// TIA Portal V17 export
// export: Created 2024-09-02T12:50:15.4689552Z, ExportSetting WithDefaults, DisplayName Totally Integrated Automation Portal, DisplayVersion V17, DisplayName TIA Portal Openness, DisplayVersion V17, DisplayName TIA Portal Version Control Interface, DisplayVersion V17, DisplayName STEP 7 Professional, DisplayVersion V17, DisplayName STEP 7 Safety, DisplayVersion V17, DisplayName WinCC Professional, DisplayVersion V17
FUNCTION "AnwFC_ZP_HMI_Management_OP70" : Void   // FC59, LAD
TITLE = HMI supply / HMI Versorgung
{ S7_Optimized_Access := 'TRUE' }
AUTHOR : OlegFuehrus
FAMILY : BA
NAME : BA
VERSION : 0.1
// stored: AutoNumber true, IsIECCheckEnabled false, SetENOAutomatically false, UDAEnableTagReadback false
   VAR_TEMP
      t_StationReady : Bool;
      tTyp : Int;
   END_VAR
   VAR_TEMP   // added for the SCL form of the ladder/FBD networks
      _w1 : Bool;
      _w2 : Bool;
   END_VAR
BEGIN

REGION Network 1: Image selection: Basic screen / Bildanwahl: Grundbild
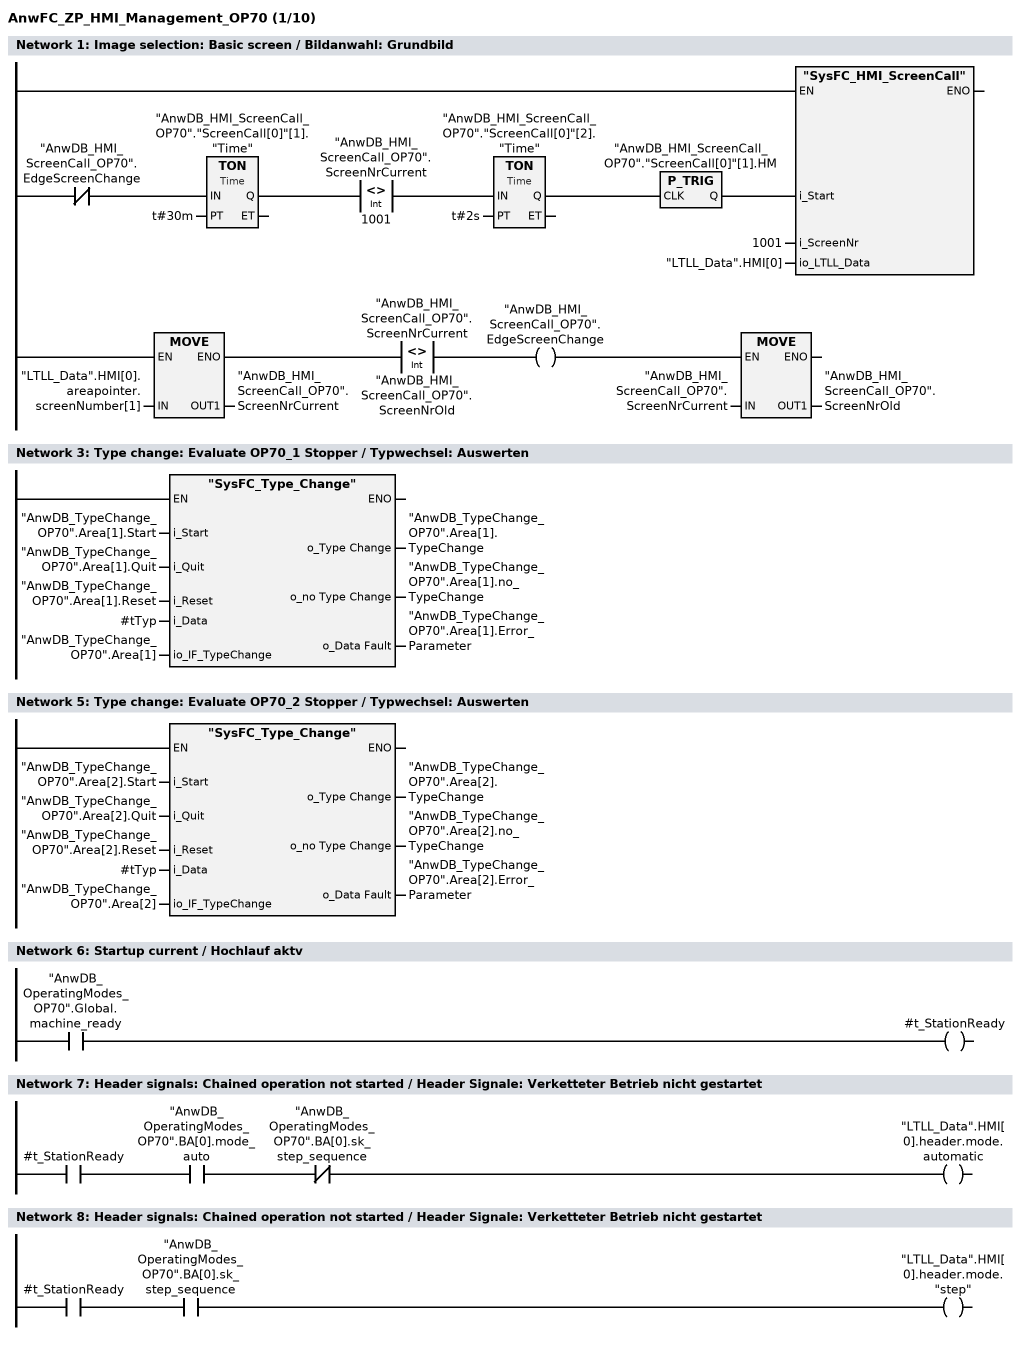
   RUNG wire#powerrail
      "SysFC_HMI_ScreenCall"(i_Start := wire#w1, i_ScreenNr := 1001, io_LTLL_Data := "LTLL_Data".HMI[0])
   END_RUNG
   RUNG wire#powerrail
      I_Contact( "AnwDB_HMI_ScreenCall_OP70".EdgeScreenChange )
      { S7_Templates := "time_type := Time" } "AnwDB_HMI_ScreenCall_OP70"."ScreenCall[0]"[1]."Time".TON(pt := t#30m, et =>)
      { S7_Templates := "SrcType := Int" } NE_Contact(in1 := "AnwDB_HMI_ScreenCall_OP70".ScreenNrCurrent, in2 := 1001)
      { S7_Templates := "time_type := Time" } "AnwDB_HMI_ScreenCall_OP70"."ScreenCall[0]"[2]."Time".TON(pt := t#2s, et =>)
      P_Trig( "AnwDB_HMI_ScreenCall_OP70"."ScreenCall[0]"[1].HM )
   END_RUNG wire#w1
   RUNG wire#powerrail
      Move(in := "LTLL_Data".HMI[0].areapointer.screenNumber[1], out1 => "AnwDB_HMI_ScreenCall_OP70".ScreenNrCurrent)
      { S7_Templates := "SrcType := Int" } NE_Contact(in1 := "AnwDB_HMI_ScreenCall_OP70".ScreenNrCurrent, in2 := "AnwDB_HMI_ScreenCall_OP70".ScreenNrOld)
      Coil( "AnwDB_HMI_ScreenCall_OP70".EdgeScreenChange )
      Move(in := "AnwDB_HMI_ScreenCall_OP70".ScreenNrCurrent, out1 => "AnwDB_HMI_ScreenCall_OP70".ScreenNrOld)
   END_RUNG
   // the same network as SCL:
   "AnwDB_HMI_ScreenCall_OP70"."ScreenCall[0]"[1]."Time".TON(IN := NOT "AnwDB_HMI_ScreenCall_OP70".EdgeScreenChange,
                           PT := t#30m);
   "AnwDB_HMI_ScreenCall_OP70"."ScreenCall[0]"[2]."Time".TON(IN := "AnwDB_HMI_ScreenCall_OP70"."ScreenCall[0]"[1]."Time".Q AND ("AnwDB_HMI_ScreenCall_OP70".ScreenNrCurrent <> 1001),
                           PT := t#2s);
   #_w1 := "AnwDB_HMI_ScreenCall_OP70"."ScreenCall[0]"[2]."Time".Q;
   #_w2 := #_w1 AND NOT "AnwDB_HMI_ScreenCall_OP70"."ScreenCall[0]"[1].HM;   // rising edge
   "AnwDB_HMI_ScreenCall_OP70"."ScreenCall[0]"[1].HM := #_w1;
   "SysFC_HMI_ScreenCall"(i_Start := #_w2, i_ScreenNr := 1001, io_LTLL_Data := "LTLL_Data".HMI[0]);
   "AnwDB_HMI_ScreenCall_OP70".ScreenNrCurrent := "LTLL_Data".HMI[0].areapointer.screenNumber[1];
   "AnwDB_HMI_ScreenCall_OP70".EdgeScreenChange := "AnwDB_HMI_ScreenCall_OP70".ScreenNrCurrent <> "AnwDB_HMI_ScreenCall_OP70".ScreenNrOld;
   IF "AnwDB_HMI_ScreenCall_OP70".EdgeScreenChange THEN
       "AnwDB_HMI_ScreenCall_OP70".ScreenNrOld := "AnwDB_HMI_ScreenCall_OP70".ScreenNrCurrent;
   END_IF;
END_REGION

REGION Network 2 (SCL): Type change: Copy type no. OP70_1 Stopper / Typwechsel: Typ-Nr. kopieren
   #tTyp := "MdsDB1_FG01_Data_SLG1_OP70".read.General."Variant Number";
END_REGION

REGION Network 3: Type change: Evaluate OP70_1 Stopper / Typwechsel: Auswerten
   RUNG wire#powerrail
      "SysFC_Type_Change"(i_Start := "AnwDB_TypeChange_OP70".Area[1].Start, i_Quit := "AnwDB_TypeChange_OP70".Area[1].Quit, i_Reset := "AnwDB_TypeChange_OP70".Area[1].Reset, i_Data := #tTyp, io_IF_TypeChange := "AnwDB_TypeChange_OP70".Area[1], "o_Type Change" => "AnwDB_TypeChange_OP70".Area[1].TypeChange, "o_no Type Change" => "AnwDB_TypeChange_OP70".Area[1].no_TypeChange, "o_Data Fault" => "AnwDB_TypeChange_OP70".Area[1].Error_Parameter)
   END_RUNG
   // the same network as SCL:
   "SysFC_Type_Change"(i_Start := "AnwDB_TypeChange_OP70".Area[1].Start,
                       i_Quit := "AnwDB_TypeChange_OP70".Area[1].Quit,
                       i_Reset := "AnwDB_TypeChange_OP70".Area[1].Reset,
                       i_Data := #tTyp,
                       io_IF_TypeChange := "AnwDB_TypeChange_OP70".Area[1],
                       "o_Type Change" => "AnwDB_TypeChange_OP70".Area[1].TypeChange,
                       "o_no Type Change" => "AnwDB_TypeChange_OP70".Area[1].no_TypeChange,
                       "o_Data Fault" => "AnwDB_TypeChange_OP70".Area[1].Error_Parameter);
END_REGION

REGION Network 4 (SCL): Type change: Copy type no. OP70_2 Stopper / Typwechsel: Typ-Nr. kopieren
   #tTyp := "MdsDB1_FG02_Data_SLG3_OP70".read.General."Variant Number";
END_REGION

REGION Network 5: Type change: Evaluate OP70_2 Stopper / Typwechsel: Auswerten
   RUNG wire#powerrail
      "SysFC_Type_Change"(i_Start := "AnwDB_TypeChange_OP70".Area[2].Start, i_Quit := "AnwDB_TypeChange_OP70".Area[2].Quit, i_Reset := "AnwDB_TypeChange_OP70".Area[2].Reset, i_Data := #tTyp, io_IF_TypeChange := "AnwDB_TypeChange_OP70".Area[2], "o_Type Change" => "AnwDB_TypeChange_OP70".Area[2].TypeChange, "o_no Type Change" => "AnwDB_TypeChange_OP70".Area[2].no_TypeChange, "o_Data Fault" => "AnwDB_TypeChange_OP70".Area[2].Error_Parameter)
   END_RUNG
   // the same network as SCL:
   "SysFC_Type_Change"(i_Start := "AnwDB_TypeChange_OP70".Area[2].Start,
                       i_Quit := "AnwDB_TypeChange_OP70".Area[2].Quit,
                       i_Reset := "AnwDB_TypeChange_OP70".Area[2].Reset,
                       i_Data := #tTyp,
                       io_IF_TypeChange := "AnwDB_TypeChange_OP70".Area[2],
                       "o_Type Change" => "AnwDB_TypeChange_OP70".Area[2].TypeChange,
                       "o_no Type Change" => "AnwDB_TypeChange_OP70".Area[2].no_TypeChange,
                       "o_Data Fault" => "AnwDB_TypeChange_OP70".Area[2].Error_Parameter);
END_REGION

REGION Network 6: Startup current / Hochlauf aktv
   RUNG wire#powerrail
      Contact( "AnwDB_OperatingModes_OP70".Global.machine_ready )
      Coil( #t_StationReady )
   END_RUNG
   // the same network as SCL:
   #t_StationReady := "AnwDB_OperatingModes_OP70".Global.machine_ready;
END_REGION

REGION Network 7: Header signals: Chained operation not started / Header Signale: Verketteter Betrieb nicht gestartet
   RUNG wire#powerrail
      Contact( #t_StationReady )
      Contact( "AnwDB_OperatingModes_OP70".BA[0].mode_auto )
      I_Contact( "AnwDB_OperatingModes_OP70".BA[0].sk_step_sequence )
      Coil( "LTLL_Data".HMI[0].header.mode.automatic )
   END_RUNG
   // the same network as SCL:
   "LTLL_Data".HMI[0].header.mode.automatic := #t_StationReady AND "AnwDB_OperatingModes_OP70".BA[0].mode_auto AND NOT "AnwDB_OperatingModes_OP70".BA[0].sk_step_sequence;
END_REGION

REGION Network 8: Header signals: Chained operation not started / Header Signale: Verketteter Betrieb nicht gestartet
   RUNG wire#powerrail
      Contact( #t_StationReady )
      Contact( "AnwDB_OperatingModes_OP70".BA[0].sk_step_sequence )
      Coil( "LTLL_Data".HMI[0].header.mode."step" )
   END_RUNG
   // the same network as SCL:
   "LTLL_Data".HMI[0].header.mode."step" := #t_StationReady AND "AnwDB_OperatingModes_OP70".BA[0].sk_step_sequence;
END_REGION

REGION Network 9: Header signals: Setup mode / Header Signale: Einrichtbetrieb
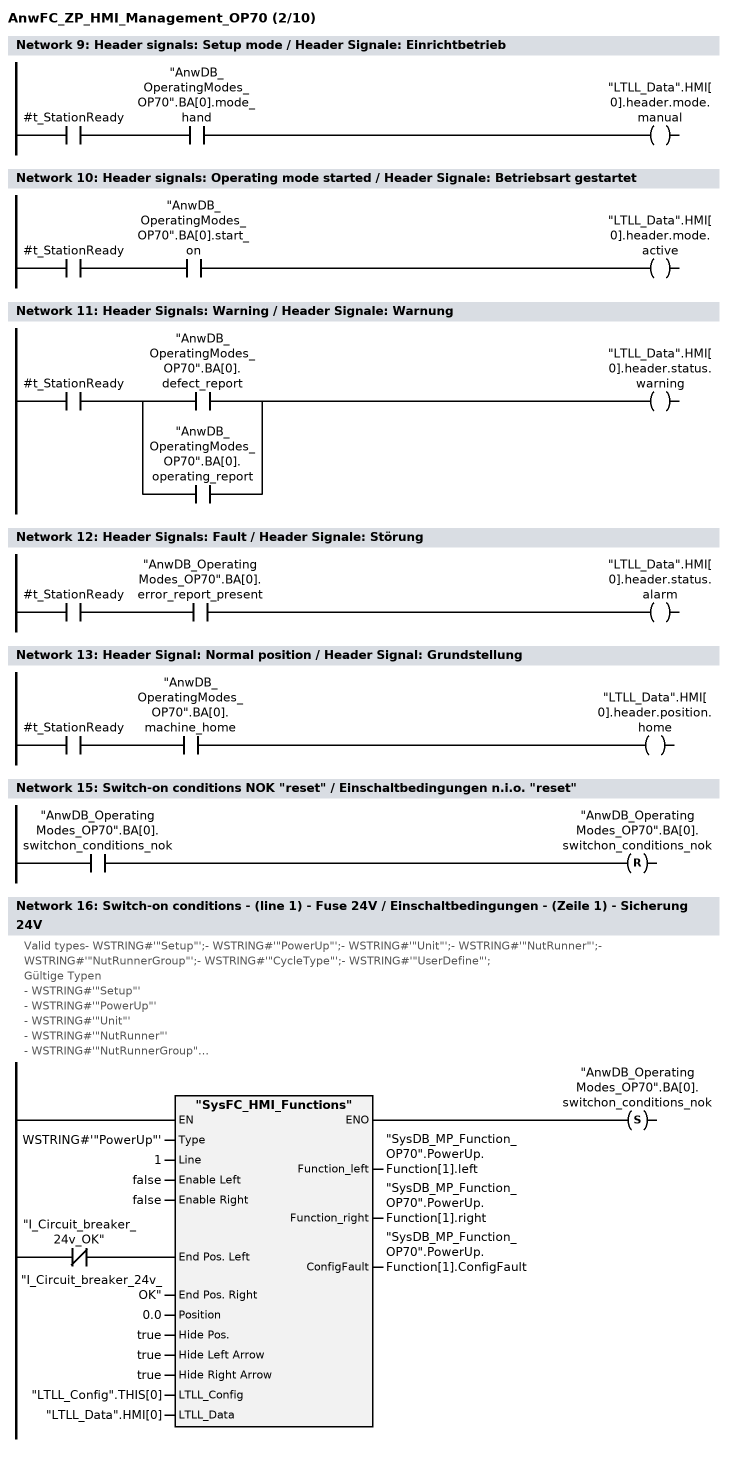
   RUNG wire#powerrail
      Contact( #t_StationReady )
      Contact( "AnwDB_OperatingModes_OP70".BA[0].mode_hand )
      Coil( "LTLL_Data".HMI[0].header.mode.manual )
   END_RUNG
   // the same network as SCL:
   "LTLL_Data".HMI[0].header.mode.manual := #t_StationReady AND "AnwDB_OperatingModes_OP70".BA[0].mode_hand;
END_REGION

REGION Network 10: Header signals: Operating mode started / Header Signale: Betriebsart gestartet
   RUNG wire#powerrail
      Contact( #t_StationReady )
      Contact( "AnwDB_OperatingModes_OP70".BA[0].start_on )
      Coil( "LTLL_Data".HMI[0].header.mode.active )
   END_RUNG
   // the same network as SCL:
   "LTLL_Data".HMI[0].header.mode.active := #t_StationReady AND "AnwDB_OperatingModes_OP70".BA[0].start_on;
END_REGION

REGION Network 11: Header Signals: Warning / Header Signale: Warnung
   RUNG wire#powerrail
      Contact( #t_StationReady )
      wire#w1
      Contact( "AnwDB_OperatingModes_OP70".BA[0].defect_report )
      wire#w2
      Coil( "LTLL_Data".HMI[0].header.status.warning )
   END_RUNG
   RUNG wire#w1
      Contact( "AnwDB_OperatingModes_OP70".BA[0].operating_report )
   END_RUNG wire#w2
   // the same network as SCL:
   "LTLL_Data".HMI[0].header.status.warning := #t_StationReady AND ("AnwDB_OperatingModes_OP70".BA[0].defect_report OR "AnwDB_OperatingModes_OP70".BA[0].operating_report);
END_REGION

REGION Network 12: Header Signals: Fault / Header Signale: Störung
   RUNG wire#powerrail
      Contact( #t_StationReady )
      Contact( "AnwDB_OperatingModes_OP70".BA[0].error_report_present )
      Coil( "LTLL_Data".HMI[0].header.status.alarm )
   END_RUNG
   // the same network as SCL:
   "LTLL_Data".HMI[0].header.status.alarm := #t_StationReady AND "AnwDB_OperatingModes_OP70".BA[0].error_report_present;
END_REGION

REGION Network 13: Header Signal: Normal position / Header Signal: Grundstellung
   RUNG wire#powerrail
      Contact( #t_StationReady )
      Contact( "AnwDB_OperatingModes_OP70".BA[0].machine_home )
      Coil( "LTLL_Data".HMI[0].header.position.home )
   END_RUNG
   // the same network as SCL:
   "LTLL_Data".HMI[0].header.position.home := #t_StationReady AND "AnwDB_OperatingModes_OP70".BA[0].machine_home;
END_REGION

REGION Network 14: ############# SO_02_002_PowerUpCondition ############## / ######################## SS_02_002_PowerUpCondition #########################
END_REGION

REGION Network 15: Switch-on conditions NOK "reset" / Einschaltbedingungen n.i.o. "reset"
   RUNG wire#powerrail
      Contact( "AnwDB_OperatingModes_OP70".BA[0].switchon_conditions_nok )
      R_Coil( "AnwDB_OperatingModes_OP70".BA[0].switchon_conditions_nok )
   END_RUNG
   // the same network as SCL:
   IF "AnwDB_OperatingModes_OP70".BA[0].switchon_conditions_nok THEN
       "AnwDB_OperatingModes_OP70".BA[0].switchon_conditions_nok := FALSE;
   END_IF;
END_REGION

REGION Network 16: Switch-on conditions - (line 1) - Fuse 24V / Einschaltbedingungen - (Zeile 1) - Sicherung 24V
   // Valid types- WSTRING#'"Setup"';- WSTRING#'"PowerUp"';- WSTRING#'"Unit"';- WSTRING#'"NutRunner"';- WSTRING#'"NutRunnerGroup"';- WSTRING#'"CycleType"';- WSTRING#'"UserDefine"';
   // Gültige Typen
   // - WSTRING#'"Setup"'
   // - WSTRING#'"PowerUp"'
   // - WSTRING#'"Unit"'
   // - WSTRING#'"NutRunner"'
   // - WSTRING#'"NutRunnerGroup"'
   // - WSTRING#'"CycleType"'
   // - WSTRING#'"UserDefine"'
   RUNG wire#powerrail
      "SysFC_HMI_Functions"("End Pos. Left" := wire#w1, "Type" := WSTRING#'"PowerUp"', Line := 1, "Enable Left" := false, "Enable Right" := false, "End Pos. Right" := "I_Circuit_breaker_24v_OK", Position := 0.0, "Hide Pos." := true, "Hide Left Arrow" := true, "Hide Right Arrow" := true, LTLL_Config := "LTLL_Config".THIS[0], LTLL_Data := "LTLL_Data".HMI[0], Function_left => "SysDB_MP_Function_OP70".PowerUp.Function[1].left, Function_right => "SysDB_MP_Function_OP70".PowerUp.Function[1].right, ConfigFault => "SysDB_MP_Function_OP70".PowerUp.Function[1].ConfigFault)
      S_Coil( "AnwDB_OperatingModes_OP70".BA[0].switchon_conditions_nok )
   END_RUNG
   RUNG wire#powerrail
      I_Contact( "I_Circuit_breaker_24v_OK" )
   END_RUNG wire#w1
   // the same network as SCL:
   "SysFC_HMI_Functions"("Type" := WSTRING#'"PowerUp"',
                         Line := 1,
                         "Enable Left" := false,
                         "Enable Right" := false,
                         "End Pos. Left" := NOT "I_Circuit_breaker_24v_OK",
                         "End Pos. Right" := "I_Circuit_breaker_24v_OK",
                         Position := 0.0,
                         "Hide Pos." := true,
                         "Hide Left Arrow" := true,
                         "Hide Right Arrow" := true,
                         LTLL_Config := "LTLL_Config".THIS[0],
                         LTLL_Data := "LTLL_Data".HMI[0],
                         Function_left => "SysDB_MP_Function_OP70".PowerUp.Function[1].left,
                         Function_right => "SysDB_MP_Function_OP70".PowerUp.Function[1].right,
                         ConfigFault => "SysDB_MP_Function_OP70".PowerUp.Function[1].ConfigFault,
                         ENO => #_w1);
   IF #_w1 THEN "AnwDB_OperatingModes_OP70".BA[0].switchon_conditions_nok := TRUE; END_IF;
END_REGION

REGION Network 17: Switch-on conditions - (line 2) - Fuse 230V / Einschaltbedingungen - (Zeile 2) - Sicherung 230V
   // Valid types- WSTRING#'"Setup"';- WSTRING#'"PowerUp"';- WSTRING#'"Unit"';- WSTRING#'"NutRunner"';- WSTRING#'"NutRunnerGroup"';- WSTRING#'"CycleType"';- WSTRING#'"UserDefine"';
   // Gültige Typen
   // - WSTRING#'"Setup"'
   // - WSTRING#'"PowerUp"'
   // - WSTRING#'"Unit"'
   // - WSTRING#'"NutRunner"'
   // - WSTRING#'"NutRunnerGroup"'
   // - WSTRING#'"CycleType"'
   // - WSTRING#'"UserDefine"'
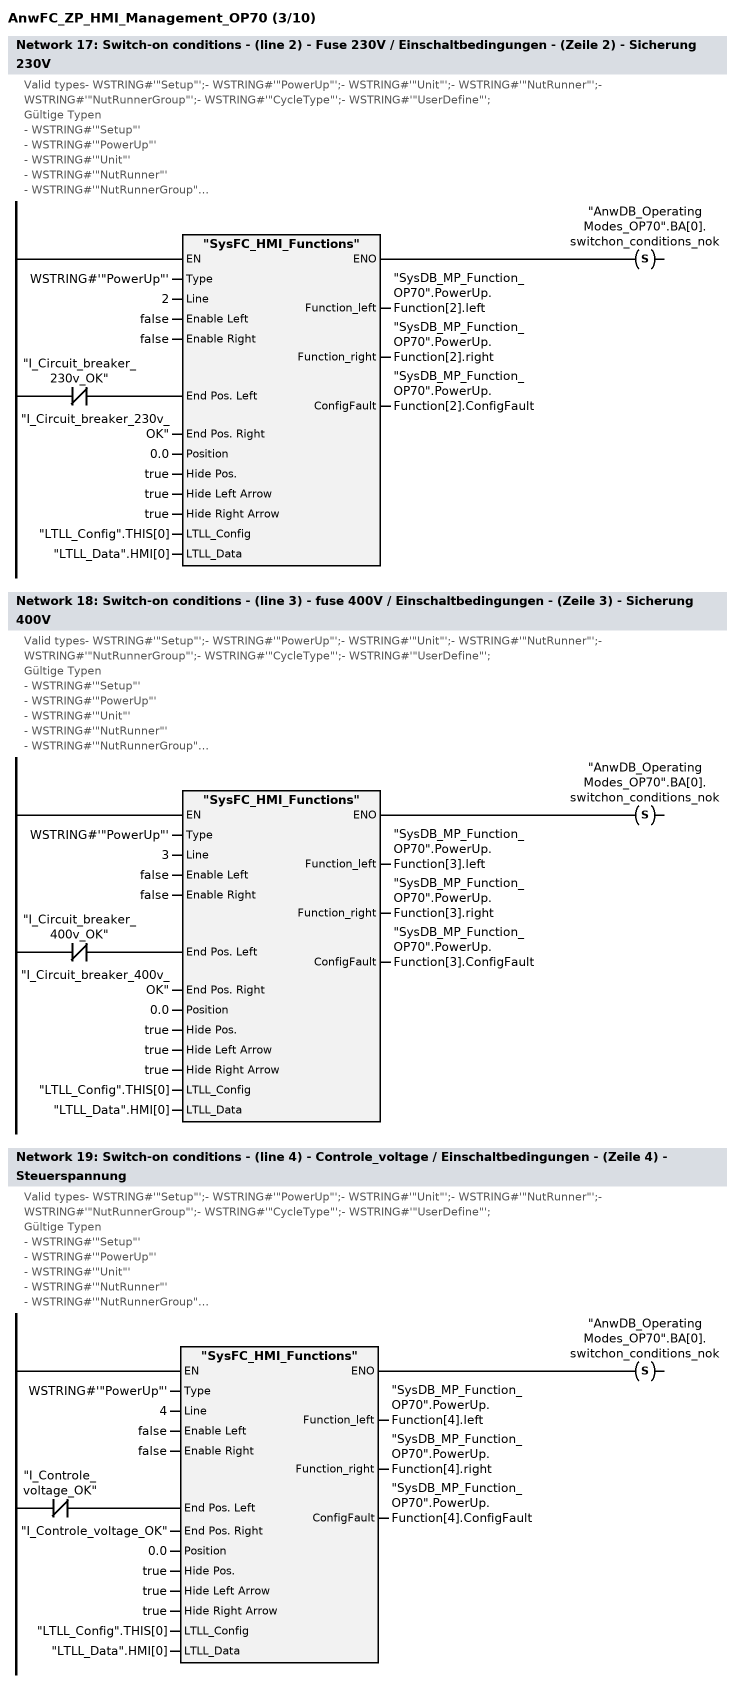
   RUNG wire#powerrail
      "SysFC_HMI_Functions"("End Pos. Left" := wire#w1, "Type" := WSTRING#'"PowerUp"', Line := 2, "Enable Left" := false, "Enable Right" := false, "End Pos. Right" := "I_Circuit_breaker_230v_OK", Position := 0.0, "Hide Pos." := true, "Hide Left Arrow" := true, "Hide Right Arrow" := true, LTLL_Config := "LTLL_Config".THIS[0], LTLL_Data := "LTLL_Data".HMI[0], Function_left => "SysDB_MP_Function_OP70".PowerUp.Function[2].left, Function_right => "SysDB_MP_Function_OP70".PowerUp.Function[2].right, ConfigFault => "SysDB_MP_Function_OP70".PowerUp.Function[2].ConfigFault)
      S_Coil( "AnwDB_OperatingModes_OP70".BA[0].switchon_conditions_nok )
   END_RUNG
   RUNG wire#powerrail
      I_Contact( "I_Circuit_breaker_230v_OK" )
   END_RUNG wire#w1
   // the same network as SCL:
   "SysFC_HMI_Functions"("Type" := WSTRING#'"PowerUp"',
                         Line := 2,
                         "Enable Left" := false,
                         "Enable Right" := false,
                         "End Pos. Left" := NOT "I_Circuit_breaker_230v_OK",
                         "End Pos. Right" := "I_Circuit_breaker_230v_OK",
                         Position := 0.0,
                         "Hide Pos." := true,
                         "Hide Left Arrow" := true,
                         "Hide Right Arrow" := true,
                         LTLL_Config := "LTLL_Config".THIS[0],
                         LTLL_Data := "LTLL_Data".HMI[0],
                         Function_left => "SysDB_MP_Function_OP70".PowerUp.Function[2].left,
                         Function_right => "SysDB_MP_Function_OP70".PowerUp.Function[2].right,
                         ConfigFault => "SysDB_MP_Function_OP70".PowerUp.Function[2].ConfigFault,
                         ENO => #_w1);
   IF #_w1 THEN "AnwDB_OperatingModes_OP70".BA[0].switchon_conditions_nok := TRUE; END_IF;
END_REGION

REGION Network 18: Switch-on conditions - (line 3) - fuse 400V / Einschaltbedingungen - (Zeile 3) - Sicherung 400V
   // Valid types- WSTRING#'"Setup"';- WSTRING#'"PowerUp"';- WSTRING#'"Unit"';- WSTRING#'"NutRunner"';- WSTRING#'"NutRunnerGroup"';- WSTRING#'"CycleType"';- WSTRING#'"UserDefine"';
   // Gültige Typen
   // - WSTRING#'"Setup"'
   // - WSTRING#'"PowerUp"'
   // - WSTRING#'"Unit"'
   // - WSTRING#'"NutRunner"'
   // - WSTRING#'"NutRunnerGroup"'
   // - WSTRING#'"CycleType"'
   // - WSTRING#'"UserDefine"'
   RUNG wire#powerrail
      "SysFC_HMI_Functions"("End Pos. Left" := wire#w1, "Type" := WSTRING#'"PowerUp"', Line := 3, "Enable Left" := false, "Enable Right" := false, "End Pos. Right" := "I_Circuit_breaker_400v_OK", Position := 0.0, "Hide Pos." := true, "Hide Left Arrow" := true, "Hide Right Arrow" := true, LTLL_Config := "LTLL_Config".THIS[0], LTLL_Data := "LTLL_Data".HMI[0], Function_left => "SysDB_MP_Function_OP70".PowerUp.Function[3].left, Function_right => "SysDB_MP_Function_OP70".PowerUp.Function[3].right, ConfigFault => "SysDB_MP_Function_OP70".PowerUp.Function[3].ConfigFault)
      S_Coil( "AnwDB_OperatingModes_OP70".BA[0].switchon_conditions_nok )
   END_RUNG
   RUNG wire#powerrail
      I_Contact( "I_Circuit_breaker_400v_OK" )
   END_RUNG wire#w1
   // the same network as SCL:
   "SysFC_HMI_Functions"("Type" := WSTRING#'"PowerUp"',
                         Line := 3,
                         "Enable Left" := false,
                         "Enable Right" := false,
                         "End Pos. Left" := NOT "I_Circuit_breaker_400v_OK",
                         "End Pos. Right" := "I_Circuit_breaker_400v_OK",
                         Position := 0.0,
                         "Hide Pos." := true,
                         "Hide Left Arrow" := true,
                         "Hide Right Arrow" := true,
                         LTLL_Config := "LTLL_Config".THIS[0],
                         LTLL_Data := "LTLL_Data".HMI[0],
                         Function_left => "SysDB_MP_Function_OP70".PowerUp.Function[3].left,
                         Function_right => "SysDB_MP_Function_OP70".PowerUp.Function[3].right,
                         ConfigFault => "SysDB_MP_Function_OP70".PowerUp.Function[3].ConfigFault,
                         ENO => #_w1);
   IF #_w1 THEN "AnwDB_OperatingModes_OP70".BA[0].switchon_conditions_nok := TRUE; END_IF;
END_REGION

REGION Network 19: Switch-on conditions - (line 4) - Controle_voltage / Einschaltbedingungen - (Zeile 4) - Steuerspannung
   // Valid types- WSTRING#'"Setup"';- WSTRING#'"PowerUp"';- WSTRING#'"Unit"';- WSTRING#'"NutRunner"';- WSTRING#'"NutRunnerGroup"';- WSTRING#'"CycleType"';- WSTRING#'"UserDefine"';
   // Gültige Typen
   // - WSTRING#'"Setup"'
   // - WSTRING#'"PowerUp"'
   // - WSTRING#'"Unit"'
   // - WSTRING#'"NutRunner"'
   // - WSTRING#'"NutRunnerGroup"'
   // - WSTRING#'"CycleType"'
   // - WSTRING#'"UserDefine"'
   RUNG wire#powerrail
      "SysFC_HMI_Functions"("End Pos. Left" := wire#w1, "Type" := WSTRING#'"PowerUp"', Line := 4, "Enable Left" := false, "Enable Right" := false, "End Pos. Right" := "I_Controle_voltage_OK", Position := 0.0, "Hide Pos." := true, "Hide Left Arrow" := true, "Hide Right Arrow" := true, LTLL_Config := "LTLL_Config".THIS[0], LTLL_Data := "LTLL_Data".HMI[0], Function_left => "SysDB_MP_Function_OP70".PowerUp.Function[4].left, Function_right => "SysDB_MP_Function_OP70".PowerUp.Function[4].right, ConfigFault => "SysDB_MP_Function_OP70".PowerUp.Function[4].ConfigFault)
      S_Coil( "AnwDB_OperatingModes_OP70".BA[0].switchon_conditions_nok )
   END_RUNG
   RUNG wire#powerrail
      I_Contact( "I_Controle_voltage_OK" )
   END_RUNG wire#w1
   // the same network as SCL:
   "SysFC_HMI_Functions"("Type" := WSTRING#'"PowerUp"',
                         Line := 4,
                         "Enable Left" := false,
                         "Enable Right" := false,
                         "End Pos. Left" := NOT "I_Controle_voltage_OK",
                         "End Pos. Right" := "I_Controle_voltage_OK",
                         Position := 0.0,
                         "Hide Pos." := true,
                         "Hide Left Arrow" := true,
                         "Hide Right Arrow" := true,
                         LTLL_Config := "LTLL_Config".THIS[0],
                         LTLL_Data := "LTLL_Data".HMI[0],
                         Function_left => "SysDB_MP_Function_OP70".PowerUp.Function[4].left,
                         Function_right => "SysDB_MP_Function_OP70".PowerUp.Function[4].right,
                         ConfigFault => "SysDB_MP_Function_OP70".PowerUp.Function[4].ConfigFault,
                         ENO => #_w1);
   IF #_w1 THEN "AnwDB_OperatingModes_OP70".BA[0].switchon_conditions_nok := TRUE; END_IF;
END_REGION

REGION Network 20: Switch-on conditions - (line 5) - Profinet / Einschaltbedingungen - (Zeile 5) - Profinet
   // Valid types- WSTRING#'"Setup"';- WSTRING#'"PowerUp"';- WSTRING#'"Unit"';- WSTRING#'"NutRunner"';- WSTRING#'"NutRunnerGroup"';- WSTRING#'"CycleType"';- WSTRING#'"UserDefine"';
   // Gültige Typen
   // - WSTRING#'"Setup"'
   // - WSTRING#'"PowerUp"'
   // - WSTRING#'"Unit"'
   // - WSTRING#'"NutRunner"'
   // - WSTRING#'"NutRunnerGroup"'
   // - WSTRING#'"CycleType"'
   // - WSTRING#'"UserDefine"'
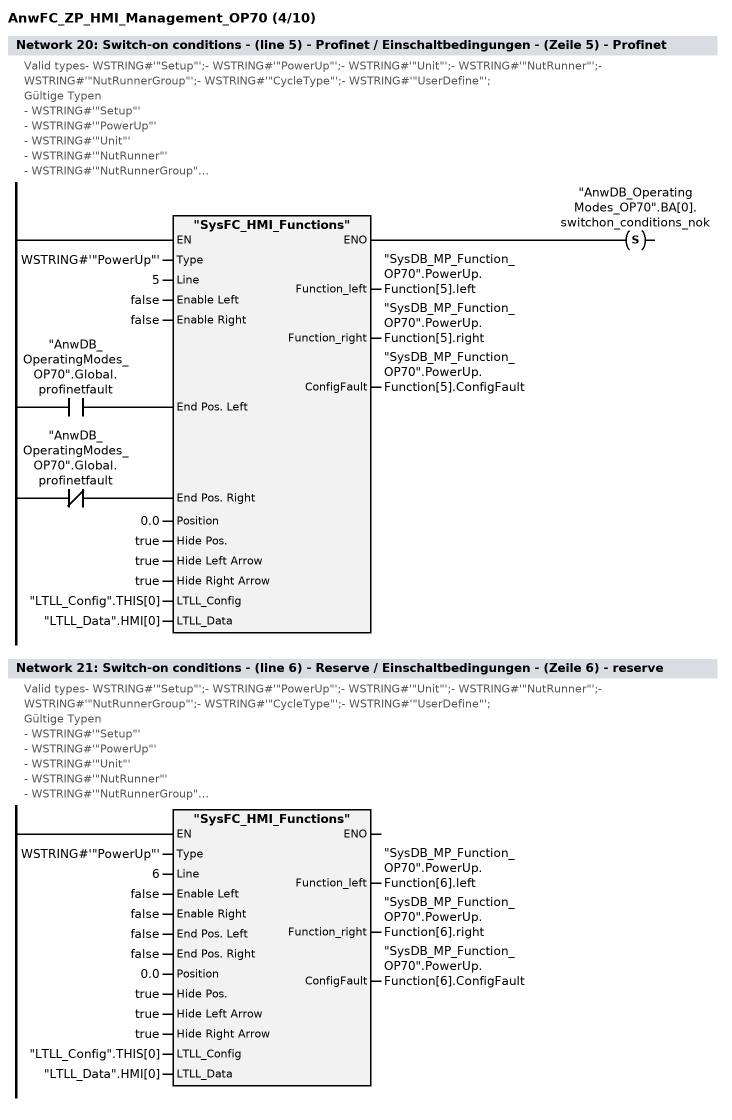
   RUNG wire#powerrail
      "SysFC_HMI_Functions"("End Pos. Left" := wire#w1, "End Pos. Right" := wire#w2, "Type" := WSTRING#'"PowerUp"', Line := 5, "Enable Left" := false, "Enable Right" := false, Position := 0.0, "Hide Pos." := true, "Hide Left Arrow" := true, "Hide Right Arrow" := true, LTLL_Config := "LTLL_Config".THIS[0], LTLL_Data := "LTLL_Data".HMI[0], Function_left => "SysDB_MP_Function_OP70".PowerUp.Function[5].left, Function_right => "SysDB_MP_Function_OP70".PowerUp.Function[5].right, ConfigFault => "SysDB_MP_Function_OP70".PowerUp.Function[5].ConfigFault)
      S_Coil( "AnwDB_OperatingModes_OP70".BA[0].switchon_conditions_nok )
   END_RUNG
   RUNG wire#powerrail
      Contact( "AnwDB_OperatingModes_OP70".Global.profinetfault )
   END_RUNG wire#w1
   RUNG wire#powerrail
      I_Contact( "AnwDB_OperatingModes_OP70".Global.profinetfault )
   END_RUNG wire#w2
   // the same network as SCL:
   "SysFC_HMI_Functions"("Type" := WSTRING#'"PowerUp"',
                         Line := 5,
                         "Enable Left" := false,
                         "Enable Right" := false,
                         "End Pos. Left" := "AnwDB_OperatingModes_OP70".Global.profinetfault,
                         "End Pos. Right" := NOT "AnwDB_OperatingModes_OP70".Global.profinetfault,
                         Position := 0.0,
                         "Hide Pos." := true,
                         "Hide Left Arrow" := true,
                         "Hide Right Arrow" := true,
                         LTLL_Config := "LTLL_Config".THIS[0],
                         LTLL_Data := "LTLL_Data".HMI[0],
                         Function_left => "SysDB_MP_Function_OP70".PowerUp.Function[5].left,
                         Function_right => "SysDB_MP_Function_OP70".PowerUp.Function[5].right,
                         ConfigFault => "SysDB_MP_Function_OP70".PowerUp.Function[5].ConfigFault,
                         ENO => #_w1);
   IF #_w1 THEN "AnwDB_OperatingModes_OP70".BA[0].switchon_conditions_nok := TRUE; END_IF;
END_REGION

REGION Network 21: Switch-on conditions - (line 6) - Reserve / Einschaltbedingungen - (Zeile 6) - reserve
   // Valid types- WSTRING#'"Setup"';- WSTRING#'"PowerUp"';- WSTRING#'"Unit"';- WSTRING#'"NutRunner"';- WSTRING#'"NutRunnerGroup"';- WSTRING#'"CycleType"';- WSTRING#'"UserDefine"';
   // Gültige Typen
   // - WSTRING#'"Setup"'
   // - WSTRING#'"PowerUp"'
   // - WSTRING#'"Unit"'
   // - WSTRING#'"NutRunner"'
   // - WSTRING#'"NutRunnerGroup"'
   // - WSTRING#'"CycleType"'
   // - WSTRING#'"UserDefine"'
   RUNG wire#powerrail
      "SysFC_HMI_Functions"("Type" := WSTRING#'"PowerUp"', Line := 6, "Enable Left" := false, "Enable Right" := false, "End Pos. Left" := false, "End Pos. Right" := false, Position := 0.0, "Hide Pos." := true, "Hide Left Arrow" := true, "Hide Right Arrow" := true, LTLL_Config := "LTLL_Config".THIS[0], LTLL_Data := "LTLL_Data".HMI[0], Function_left => "SysDB_MP_Function_OP70".PowerUp.Function[6].left, Function_right => "SysDB_MP_Function_OP70".PowerUp.Function[6].right, ConfigFault => "SysDB_MP_Function_OP70".PowerUp.Function[6].ConfigFault)
   END_RUNG
   // the same network as SCL:
   "SysFC_HMI_Functions"("Type" := WSTRING#'"PowerUp"',
                         Line := 6,
                         "Enable Left" := false,
                         "Enable Right" := false,
                         "End Pos. Left" := false,
                         "End Pos. Right" := false,
                         Position := 0.0,
                         "Hide Pos." := true,
                         "Hide Left Arrow" := true,
                         "Hide Right Arrow" := true,
                         LTLL_Config := "LTLL_Config".THIS[0],
                         LTLL_Data := "LTLL_Data".HMI[0],
                         Function_left => "SysDB_MP_Function_OP70".PowerUp.Function[6].left,
                         Function_right => "SysDB_MP_Function_OP70".PowerUp.Function[6].right,
                         ConfigFault => "SysDB_MP_Function_OP70".PowerUp.Function[6].ConfigFault);
END_REGION

REGION Network 22: Switch-on conditions - (line 7) - Safety door OP40 / Einschaltbedingungen - (Zeile 7) - Schutztüren OP40
   // Valid types- WSTRING#'"Setup"';- WSTRING#'"PowerUp"';- WSTRING#'"Unit"';- WSTRING#'"NutRunner"';- WSTRING#'"NutRunnerGroup"';- WSTRING#'"CycleType"';- WSTRING#'"UserDefine"';
   // Gültige Typen
   // - WSTRING#'"Setup"'
   // - WSTRING#'"PowerUp"'
   // - WSTRING#'"Unit"'
   // - WSTRING#'"NutRunner"'
   // - WSTRING#'"NutRunnerGroup"'
   // - WSTRING#'"CycleType"'
   // - WSTRING#'"UserDefine"'
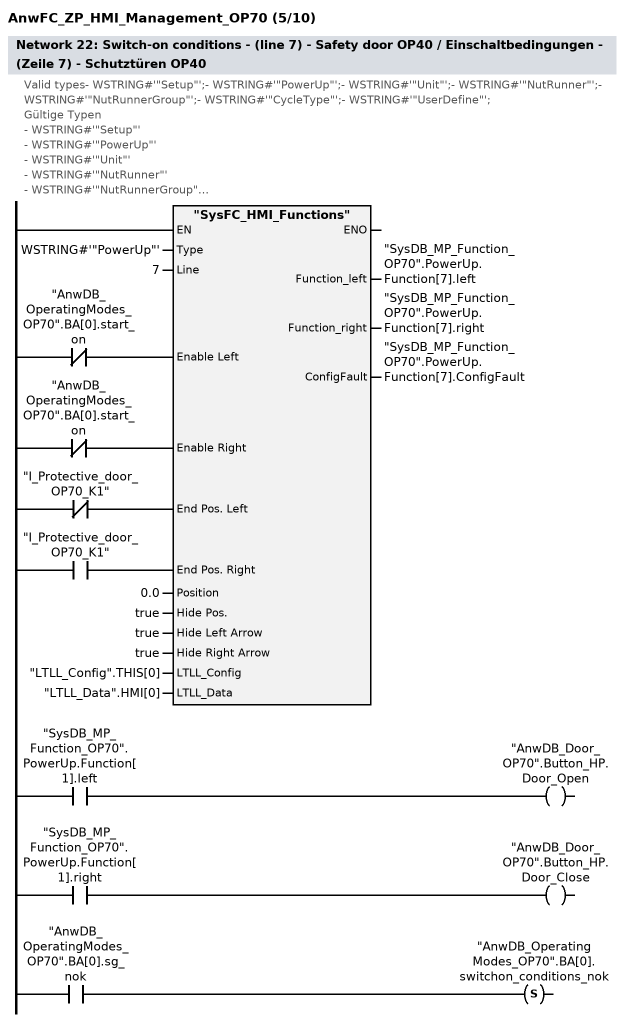
   RUNG wire#powerrail
      "SysFC_HMI_Functions"("Enable Left" := wire#w1, "Enable Right" := wire#w2, "End Pos. Left" := wire#w3, "End Pos. Right" := wire#w4, "Type" := WSTRING#'"PowerUp"', Line := 7, Position := 0.0, "Hide Pos." := true, "Hide Left Arrow" := true, "Hide Right Arrow" := true, LTLL_Config := "LTLL_Config".THIS[0], LTLL_Data := "LTLL_Data".HMI[0], Function_left => "SysDB_MP_Function_OP70".PowerUp.Function[7].left, Function_right => "SysDB_MP_Function_OP70".PowerUp.Function[7].right, ConfigFault => "SysDB_MP_Function_OP70".PowerUp.Function[7].ConfigFault)
   END_RUNG
   RUNG wire#powerrail
      I_Contact( "AnwDB_OperatingModes_OP70".BA[0].start_on )
   END_RUNG wire#w1
   RUNG wire#powerrail
      I_Contact( "AnwDB_OperatingModes_OP70".BA[0].start_on )
   END_RUNG wire#w2
   RUNG wire#powerrail
      I_Contact( "I_Protective_door_OP70_K1" )
   END_RUNG wire#w3
   RUNG wire#powerrail
      Contact( "I_Protective_door_OP70_K1" )
   END_RUNG wire#w4
   RUNG wire#powerrail
      Contact( "SysDB_MP_Function_OP70".PowerUp.Function[1].left )
      Coil( "AnwDB_Door_OP70".Button_HP.Door_Open )
   END_RUNG
   RUNG wire#powerrail
      Contact( "SysDB_MP_Function_OP70".PowerUp.Function[1].right )
      Coil( "AnwDB_Door_OP70".Button_HP.Door_Close )
   END_RUNG
   RUNG wire#powerrail
      Contact( "AnwDB_OperatingModes_OP70".BA[0].sg_nok )
      S_Coil( "AnwDB_OperatingModes_OP70".BA[0].switchon_conditions_nok )
   END_RUNG
   // the same network as SCL:
   "SysFC_HMI_Functions"("Type" := WSTRING#'"PowerUp"',
                         Line := 7,
                         "Enable Left" := NOT "AnwDB_OperatingModes_OP70".BA[0].start_on,
                         "Enable Right" := NOT "AnwDB_OperatingModes_OP70".BA[0].start_on,
                         "End Pos. Left" := NOT "I_Protective_door_OP70_K1",
                         "End Pos. Right" := "I_Protective_door_OP70_K1",
                         Position := 0.0,
                         "Hide Pos." := true,
                         "Hide Left Arrow" := true,
                         "Hide Right Arrow" := true,
                         LTLL_Config := "LTLL_Config".THIS[0],
                         LTLL_Data := "LTLL_Data".HMI[0],
                         Function_left => "SysDB_MP_Function_OP70".PowerUp.Function[7].left,
                         Function_right => "SysDB_MP_Function_OP70".PowerUp.Function[7].right,
                         ConfigFault => "SysDB_MP_Function_OP70".PowerUp.Function[7].ConfigFault);
   "AnwDB_Door_OP70".Button_HP.Door_Open := "SysDB_MP_Function_OP70".PowerUp.Function[1].left;
   "AnwDB_Door_OP70".Button_HP.Door_Close := "SysDB_MP_Function_OP70".PowerUp.Function[1].right;
   IF "AnwDB_OperatingModes_OP70".BA[0].sg_nok THEN
       "AnwDB_OperatingModes_OP70".BA[0].switchon_conditions_nok := TRUE;
   END_IF;
END_REGION

REGION Network 23: Switch-on conditions - (line 8) - Pneumatics OP40 / Einschaltbedingungen - (Zeile 8) - Pneumatik OP40
   // Valid types- WSTRING#'"Setup"';- WSTRING#'"PowerUp"';- WSTRING#'"Unit"';- WSTRING#'"NutRunner"';- WSTRING#'"NutRunnerGroup"';- WSTRING#'"CycleType"';- WSTRING#'"UserDefine"';
   // Gültige Typen
   // - WSTRING#'"Setup"'
   // - WSTRING#'"PowerUp"'
   // - WSTRING#'"Unit"'
   // - WSTRING#'"NutRunner"'
   // - WSTRING#'"NutRunnerGroup"'
   // - WSTRING#'"CycleType"'
   // - WSTRING#'"UserDefine"'
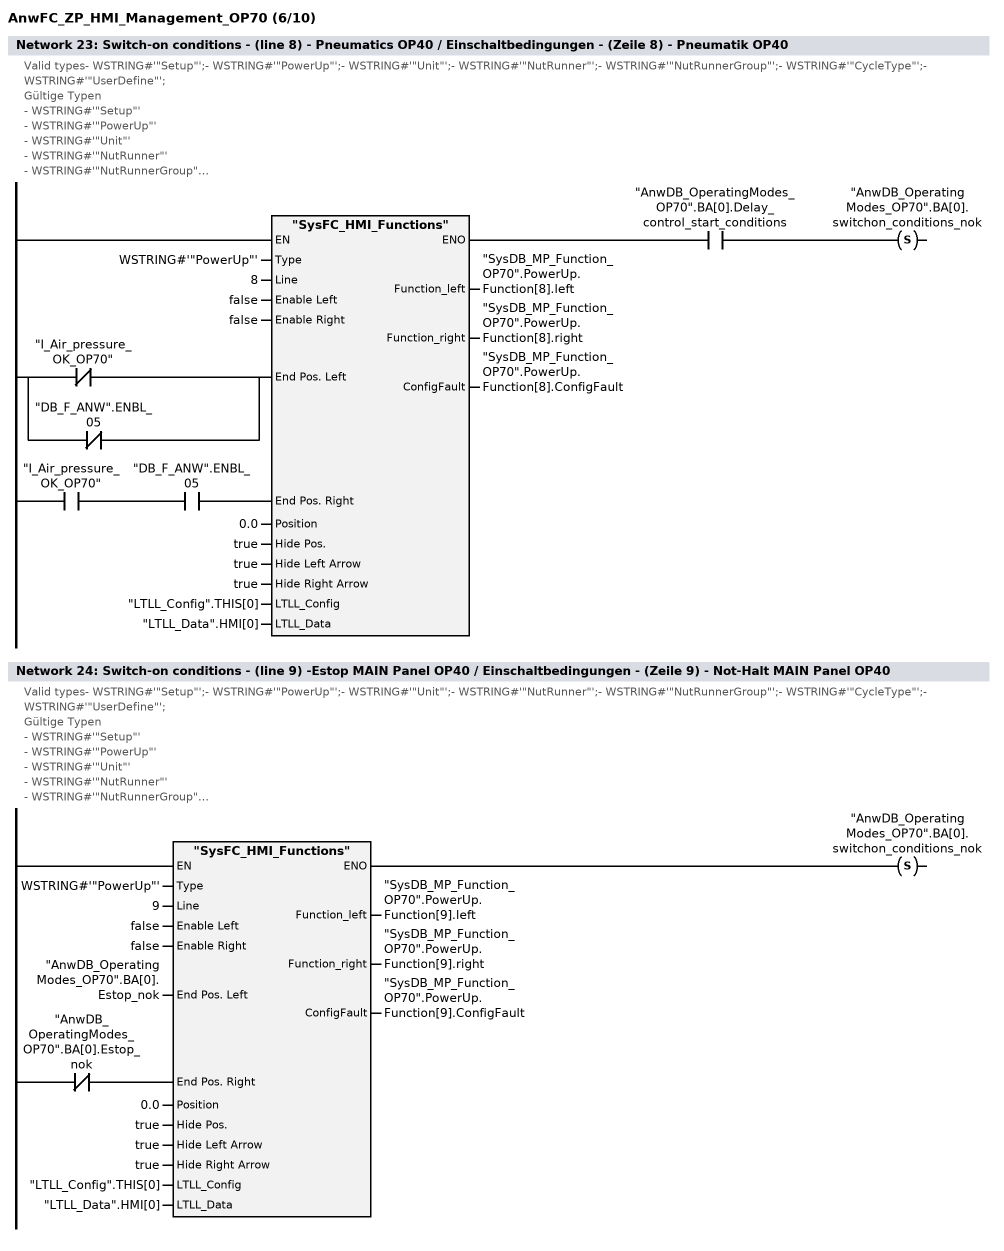
   RUNG wire#powerrail
      "SysFC_HMI_Functions"("End Pos. Left" := wire#w1, "End Pos. Right" := wire#w2, "Type" := WSTRING#'"PowerUp"', Line := 8, "Enable Left" := false, "Enable Right" := false, Position := 0.0, "Hide Pos." := true, "Hide Left Arrow" := true, "Hide Right Arrow" := true, LTLL_Config := "LTLL_Config".THIS[0], LTLL_Data := "LTLL_Data".HMI[0], Function_left => "SysDB_MP_Function_OP70".PowerUp.Function[8].left, Function_right => "SysDB_MP_Function_OP70".PowerUp.Function[8].right, ConfigFault => "SysDB_MP_Function_OP70".PowerUp.Function[8].ConfigFault)
      Contact( "AnwDB_OperatingModes_OP70".BA[0].Delay_control_start_conditions )
      S_Coil( "AnwDB_OperatingModes_OP70".BA[0].switchon_conditions_nok )
   END_RUNG
   RUNG wire#powerrail
      I_Contact( "I_Air_pressure_OK_OP70" )
   END_RUNG wire#w1
   RUNG wire#powerrail
      I_Contact( "DB_F_ANW".ENBL_05 )
   END_RUNG wire#w1
   RUNG wire#powerrail
      Contact( "I_Air_pressure_OK_OP70" )
      Contact( "DB_F_ANW".ENBL_05 )
   END_RUNG wire#w2
   // the same network as SCL:
   "SysFC_HMI_Functions"("Type" := WSTRING#'"PowerUp"',
                         Line := 8,
                         "Enable Left" := false,
                         "Enable Right" := false,
                         "End Pos. Left" := NOT "I_Air_pressure_OK_OP70" OR NOT "DB_F_ANW".ENBL_05,
                         "End Pos. Right" := "I_Air_pressure_OK_OP70" AND "DB_F_ANW".ENBL_05,
                         Position := 0.0,
                         "Hide Pos." := true,
                         "Hide Left Arrow" := true,
                         "Hide Right Arrow" := true,
                         LTLL_Config := "LTLL_Config".THIS[0],
                         LTLL_Data := "LTLL_Data".HMI[0],
                         Function_left => "SysDB_MP_Function_OP70".PowerUp.Function[8].left,
                         Function_right => "SysDB_MP_Function_OP70".PowerUp.Function[8].right,
                         ConfigFault => "SysDB_MP_Function_OP70".PowerUp.Function[8].ConfigFault,
                         ENO => #_w1);
   IF #_w1 AND "AnwDB_OperatingModes_OP70".BA[0].Delay_control_start_conditions THEN
       "AnwDB_OperatingModes_OP70".BA[0].switchon_conditions_nok := TRUE;
   END_IF;
END_REGION

REGION Network 24: Switch-on conditions - (line 9) -Estop MAIN Panel OP40 / Einschaltbedingungen - (Zeile 9) - Not-Halt MAIN Panel OP40
   // Valid types- WSTRING#'"Setup"';- WSTRING#'"PowerUp"';- WSTRING#'"Unit"';- WSTRING#'"NutRunner"';- WSTRING#'"NutRunnerGroup"';- WSTRING#'"CycleType"';- WSTRING#'"UserDefine"';
   // Gültige Typen
   // - WSTRING#'"Setup"'
   // - WSTRING#'"PowerUp"'
   // - WSTRING#'"Unit"'
   // - WSTRING#'"NutRunner"'
   // - WSTRING#'"NutRunnerGroup"'
   // - WSTRING#'"CycleType"'
   // - WSTRING#'"UserDefine"'
   RUNG wire#powerrail
      "SysFC_HMI_Functions"("End Pos. Right" := wire#w1, "Type" := WSTRING#'"PowerUp"', Line := 9, "Enable Left" := false, "Enable Right" := false, "End Pos. Left" := "AnwDB_OperatingModes_OP70".BA[0].Estop_nok, Position := 0.0, "Hide Pos." := true, "Hide Left Arrow" := true, "Hide Right Arrow" := true, LTLL_Config := "LTLL_Config".THIS[0], LTLL_Data := "LTLL_Data".HMI[0], Function_left => "SysDB_MP_Function_OP70".PowerUp.Function[9].left, Function_right => "SysDB_MP_Function_OP70".PowerUp.Function[9].right, ConfigFault => "SysDB_MP_Function_OP70".PowerUp.Function[9].ConfigFault)
      S_Coil( "AnwDB_OperatingModes_OP70".BA[0].switchon_conditions_nok )
   END_RUNG
   RUNG wire#powerrail
      I_Contact( "AnwDB_OperatingModes_OP70".BA[0].Estop_nok )
   END_RUNG wire#w1
   // the same network as SCL:
   "SysFC_HMI_Functions"("Type" := WSTRING#'"PowerUp"',
                         Line := 9,
                         "Enable Left" := false,
                         "Enable Right" := false,
                         "End Pos. Left" := "AnwDB_OperatingModes_OP70".BA[0].Estop_nok,
                         "End Pos. Right" := NOT "AnwDB_OperatingModes_OP70".BA[0].Estop_nok,
                         Position := 0.0,
                         "Hide Pos." := true,
                         "Hide Left Arrow" := true,
                         "Hide Right Arrow" := true,
                         LTLL_Config := "LTLL_Config".THIS[0],
                         LTLL_Data := "LTLL_Data".HMI[0],
                         Function_left => "SysDB_MP_Function_OP70".PowerUp.Function[9].left,
                         Function_right => "SysDB_MP_Function_OP70".PowerUp.Function[9].right,
                         ConfigFault => "SysDB_MP_Function_OP70".PowerUp.Function[9].ConfigFault,
                         ENO => #_w1);
   IF #_w1 THEN "AnwDB_OperatingModes_OP70".BA[0].switchon_conditions_nok := TRUE; END_IF;
END_REGION

REGION Network 25: Switch-on conditions - (line 10) - Reserve / Einschaltbedingungen - (Zeile 10) - reserve
   // Valid types- WSTRING#'"Setup"';- WSTRING#'"PowerUp"';- WSTRING#'"Unit"';- WSTRING#'"NutRunner"';- WSTRING#'"NutRunnerGroup"';- WSTRING#'"CycleType"';- WSTRING#'"UserDefine"';
   // Gültige Typen
   // - WSTRING#'"Setup"'
   // - WSTRING#'"PowerUp"'
   // - WSTRING#'"Unit"'
   // - WSTRING#'"NutRunner"'
   // - WSTRING#'"NutRunnerGroup"'
   // - WSTRING#'"CycleType"'
   // - WSTRING#'"UserDefine"'
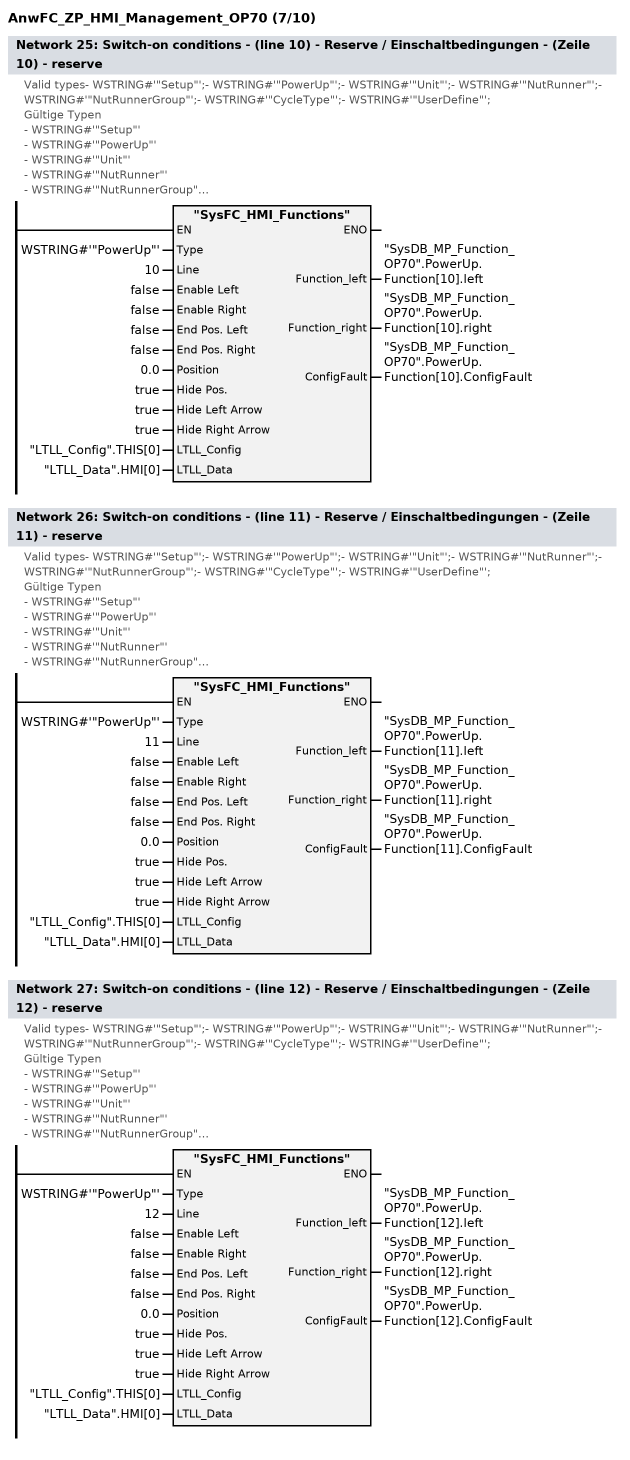
   RUNG wire#powerrail
      "SysFC_HMI_Functions"("Type" := WSTRING#'"PowerUp"', Line := 10, "Enable Left" := false, "Enable Right" := false, "End Pos. Left" := false, "End Pos. Right" := false, Position := 0.0, "Hide Pos." := true, "Hide Left Arrow" := true, "Hide Right Arrow" := true, LTLL_Config := "LTLL_Config".THIS[0], LTLL_Data := "LTLL_Data".HMI[0], Function_left => "SysDB_MP_Function_OP70".PowerUp.Function[10].left, Function_right => "SysDB_MP_Function_OP70".PowerUp.Function[10].right, ConfigFault => "SysDB_MP_Function_OP70".PowerUp.Function[10].ConfigFault)
   END_RUNG
   // the same network as SCL:
   "SysFC_HMI_Functions"("Type" := WSTRING#'"PowerUp"',
                         Line := 10,
                         "Enable Left" := false,
                         "Enable Right" := false,
                         "End Pos. Left" := false,
                         "End Pos. Right" := false,
                         Position := 0.0,
                         "Hide Pos." := true,
                         "Hide Left Arrow" := true,
                         "Hide Right Arrow" := true,
                         LTLL_Config := "LTLL_Config".THIS[0],
                         LTLL_Data := "LTLL_Data".HMI[0],
                         Function_left => "SysDB_MP_Function_OP70".PowerUp.Function[10].left,
                         Function_right => "SysDB_MP_Function_OP70".PowerUp.Function[10].right,
                         ConfigFault => "SysDB_MP_Function_OP70".PowerUp.Function[10].ConfigFault);
END_REGION

REGION Network 26: Switch-on conditions - (line 11) - Reserve / Einschaltbedingungen - (Zeile 11) - reserve
   // Valid types- WSTRING#'"Setup"';- WSTRING#'"PowerUp"';- WSTRING#'"Unit"';- WSTRING#'"NutRunner"';- WSTRING#'"NutRunnerGroup"';- WSTRING#'"CycleType"';- WSTRING#'"UserDefine"';
   // Gültige Typen
   // - WSTRING#'"Setup"'
   // - WSTRING#'"PowerUp"'
   // - WSTRING#'"Unit"'
   // - WSTRING#'"NutRunner"'
   // - WSTRING#'"NutRunnerGroup"'
   // - WSTRING#'"CycleType"'
   // - WSTRING#'"UserDefine"'
   RUNG wire#powerrail
      "SysFC_HMI_Functions"("Type" := WSTRING#'"PowerUp"', Line := 11, "Enable Left" := false, "Enable Right" := false, "End Pos. Left" := false, "End Pos. Right" := false, Position := 0.0, "Hide Pos." := true, "Hide Left Arrow" := true, "Hide Right Arrow" := true, LTLL_Config := "LTLL_Config".THIS[0], LTLL_Data := "LTLL_Data".HMI[0], Function_left => "SysDB_MP_Function_OP70".PowerUp.Function[11].left, Function_right => "SysDB_MP_Function_OP70".PowerUp.Function[11].right, ConfigFault => "SysDB_MP_Function_OP70".PowerUp.Function[11].ConfigFault)
   END_RUNG
   // the same network as SCL:
   "SysFC_HMI_Functions"("Type" := WSTRING#'"PowerUp"',
                         Line := 11,
                         "Enable Left" := false,
                         "Enable Right" := false,
                         "End Pos. Left" := false,
                         "End Pos. Right" := false,
                         Position := 0.0,
                         "Hide Pos." := true,
                         "Hide Left Arrow" := true,
                         "Hide Right Arrow" := true,
                         LTLL_Config := "LTLL_Config".THIS[0],
                         LTLL_Data := "LTLL_Data".HMI[0],
                         Function_left => "SysDB_MP_Function_OP70".PowerUp.Function[11].left,
                         Function_right => "SysDB_MP_Function_OP70".PowerUp.Function[11].right,
                         ConfigFault => "SysDB_MP_Function_OP70".PowerUp.Function[11].ConfigFault);
END_REGION

REGION Network 27: Switch-on conditions - (line 12) - Reserve / Einschaltbedingungen - (Zeile 12) - reserve
   // Valid types- WSTRING#'"Setup"';- WSTRING#'"PowerUp"';- WSTRING#'"Unit"';- WSTRING#'"NutRunner"';- WSTRING#'"NutRunnerGroup"';- WSTRING#'"CycleType"';- WSTRING#'"UserDefine"';
   // Gültige Typen
   // - WSTRING#'"Setup"'
   // - WSTRING#'"PowerUp"'
   // - WSTRING#'"Unit"'
   // - WSTRING#'"NutRunner"'
   // - WSTRING#'"NutRunnerGroup"'
   // - WSTRING#'"CycleType"'
   // - WSTRING#'"UserDefine"'
   RUNG wire#powerrail
      "SysFC_HMI_Functions"("Type" := WSTRING#'"PowerUp"', Line := 12, "Enable Left" := false, "Enable Right" := false, "End Pos. Left" := false, "End Pos. Right" := false, Position := 0.0, "Hide Pos." := true, "Hide Left Arrow" := true, "Hide Right Arrow" := true, LTLL_Config := "LTLL_Config".THIS[0], LTLL_Data := "LTLL_Data".HMI[0], Function_left => "SysDB_MP_Function_OP70".PowerUp.Function[12].left, Function_right => "SysDB_MP_Function_OP70".PowerUp.Function[12].right, ConfigFault => "SysDB_MP_Function_OP70".PowerUp.Function[12].ConfigFault)
   END_RUNG
   // the same network as SCL:
   "SysFC_HMI_Functions"("Type" := WSTRING#'"PowerUp"',
                         Line := 12,
                         "Enable Left" := false,
                         "Enable Right" := false,
                         "End Pos. Left" := false,
                         "End Pos. Right" := false,
                         Position := 0.0,
                         "Hide Pos." := true,
                         "Hide Left Arrow" := true,
                         "Hide Right Arrow" := true,
                         LTLL_Config := "LTLL_Config".THIS[0],
                         LTLL_Data := "LTLL_Data".HMI[0],
                         Function_left => "SysDB_MP_Function_OP70".PowerUp.Function[12].left,
                         Function_right => "SysDB_MP_Function_OP70".PowerUp.Function[12].right,
                         ConfigFault => "SysDB_MP_Function_OP70".PowerUp.Function[12].ConfigFault);
END_REGION

REGION Network 28: ############# OO_30_000_SERVICE ##############
END_REGION

REGION Network 29: Jump Ouf Of Service Screen
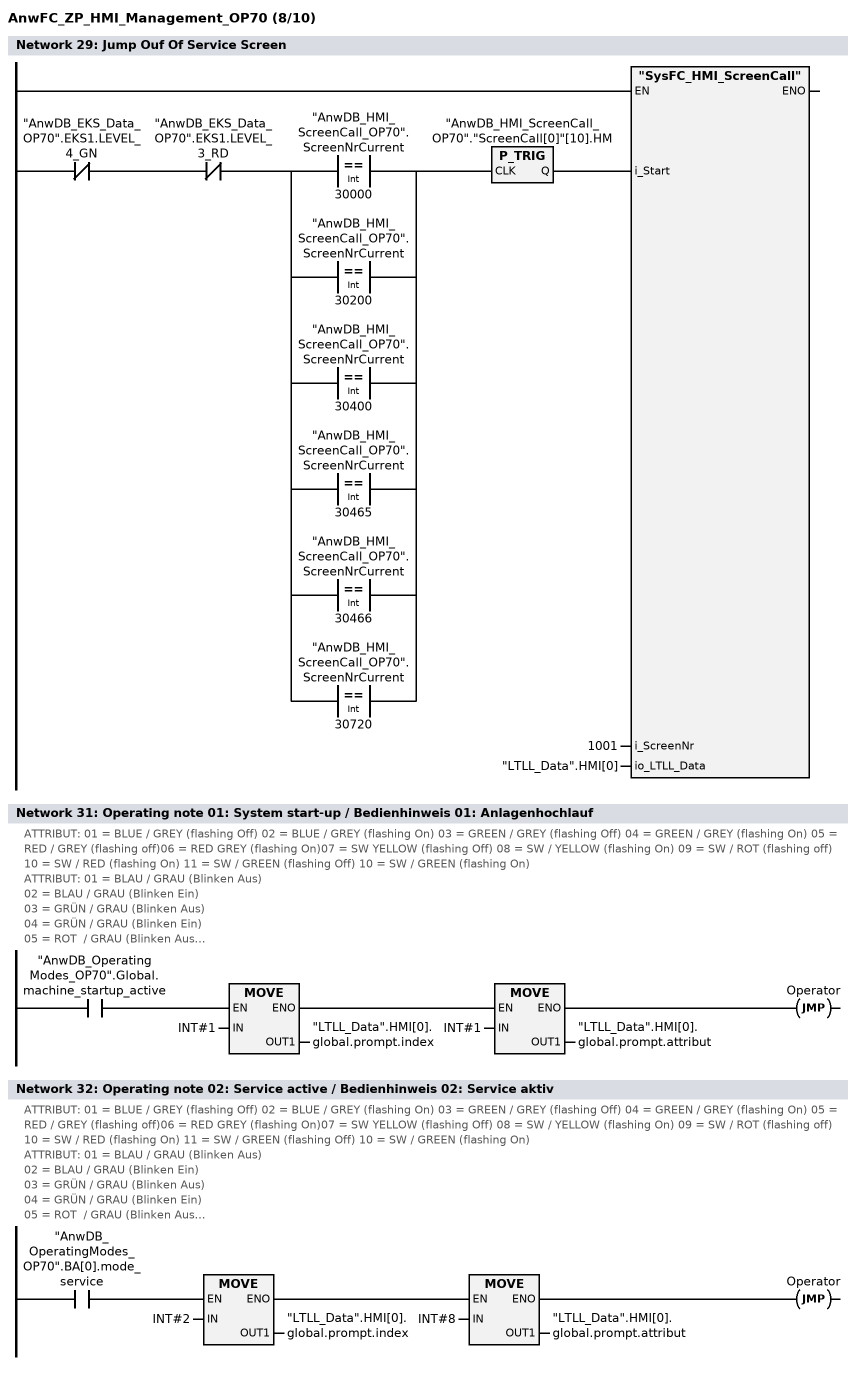
   RUNG wire#powerrail
      "SysFC_HMI_ScreenCall"(i_Start := wire#w3, i_ScreenNr := 1001, io_LTLL_Data := "LTLL_Data".HMI[0])
   END_RUNG
   RUNG wire#powerrail
      I_Contact( "AnwDB_EKS_Data_OP70".EKS1.LEVEL_4_GN )
      I_Contact( "AnwDB_EKS_Data_OP70".EKS1.LEVEL_3_RD )
      wire#w1
      { S7_Templates := "SrcType := Int" } EQ_Contact(in1 := "AnwDB_HMI_ScreenCall_OP70".ScreenNrCurrent, in2 := 30000)
      wire#w2
      P_Trig( "AnwDB_HMI_ScreenCall_OP70"."ScreenCall[0]"[10].HM )
   END_RUNG wire#w3
   RUNG wire#w1
      { S7_Templates := "SrcType := Int" } EQ_Contact(in1 := "AnwDB_HMI_ScreenCall_OP70".ScreenNrCurrent, in2 := 30200)
   END_RUNG wire#w2
   RUNG wire#w1
      { S7_Templates := "SrcType := Int" } EQ_Contact(in1 := "AnwDB_HMI_ScreenCall_OP70".ScreenNrCurrent, in2 := 30400)
   END_RUNG wire#w2
   RUNG wire#w1
      { S7_Templates := "SrcType := Int" } EQ_Contact(in1 := "AnwDB_HMI_ScreenCall_OP70".ScreenNrCurrent, in2 := 30465)
   END_RUNG wire#w2
   RUNG wire#w1
      { S7_Templates := "SrcType := Int" } EQ_Contact(in1 := "AnwDB_HMI_ScreenCall_OP70".ScreenNrCurrent, in2 := 30466)
   END_RUNG wire#w2
   RUNG wire#w1
      { S7_Templates := "SrcType := Int" } EQ_Contact(in1 := "AnwDB_HMI_ScreenCall_OP70".ScreenNrCurrent, in2 := 30720)
   END_RUNG wire#w2
   // the same network as SCL:
   #_w1 := NOT "AnwDB_EKS_Data_OP70".EKS1.LEVEL_4_GN AND NOT "AnwDB_EKS_Data_OP70".EKS1.LEVEL_3_RD AND (("AnwDB_HMI_ScreenCall_OP70".ScreenNrCurrent = 30000) OR ("AnwDB_HMI_ScreenCall_OP70".ScreenNrCurrent = 30200) OR ("AnwDB_HMI_ScreenCall_OP70".ScreenNrCurrent = 30400) OR ("AnwDB_HMI_ScreenCall_OP70".ScreenNrCurrent = 30465) OR ("AnwDB_HMI_ScreenCall_OP70".ScreenNrCurrent = 30466) OR ("AnwDB_HMI_ScreenCall_OP70".ScreenNrCurrent = 30720));
   #_w2 := #_w1 AND NOT "AnwDB_HMI_ScreenCall_OP70"."ScreenCall[0]"[10].HM;   // rising edge
   "AnwDB_HMI_ScreenCall_OP70"."ScreenCall[0]"[10].HM := #_w1;
   "SysFC_HMI_ScreenCall"(i_Start := #_w2, i_ScreenNr := 1001, io_LTLL_Data := "LTLL_Data".HMI[0]);
END_REGION

REGION Network 30: ############# SO_00_000_OperatorPrompt ############## / ######################## SO_00_000_OperatorPrompt ###########################
END_REGION

REGION Network 31: Operating note 01: System start-up / Bedienhinweis 01: Anlagenhochlauf
   // ATTRIBUT: 01 = BLUE / GREY (flashing Off) 02 = BLUE / GREY (flashing On) 03 = GREEN / GREY (flashing Off) 04 = GREEN / GREY (flashing On) 05 = RED / GREY (flashing off)06 = RED GREY (flashing On)07 = SW YELLOW (flashing Off) 08 = SW / YELLOW (flashing On) 09 = SW / ROT (flashing off) 10 = SW / RED (flashing On) 11 = SW / GREEN (flashing Off) 10 = SW / GREEN (flashing On)
   // ATTRIBUT: 01 = BLAU / GRAU (Blinken Aus)
   //           02 = BLAU / GRAU (Blinken Ein)
   //           03 = GRÜN / GRAU (Blinken Aus)
   //           04 = GRÜN / GRAU (Blinken Ein)
   //           05 = ROT  / GRAU (Blinken Aus)
   //           06 = ROT  / GRAU (Blinken Ein)
   //           07 = SW   / GELB (Blinken Aus)
   //           08 = SW   / GELB (Blinken Ein)
   //           09 = SW   / ROT  (Blinken Aus)
   //           10 = SW   / ROT  (Blinken Ein)
   //           11 = SW   / GRÜN (Blinken Aus)
   //           10 = SW   / GRÜN (Blinken Ein)
   RUNG wire#powerrail
      Contact( "AnwDB_OperatingModes_OP70".Global.machine_startup_active )
      { S7_GenerateENO := "TRUE" } Move(in := INT#1, out1 => "LTLL_Data".HMI[0].global.prompt.index)
      { S7_GenerateENO := "TRUE" } Move(in := INT#1, out1 => "LTLL_Data".HMI[0].global.prompt.attribut)
      JumpCoil( Operator )
   END_RUNG
   // the same network as SCL:
   // ENO of a box is taken as its EN; it also drops when the box reports an error
   IF "AnwDB_OperatingModes_OP70".Global.machine_startup_active THEN
       "LTLL_Data".HMI[0].global.prompt.index := INT#1;
       "LTLL_Data".HMI[0].global.prompt.attribut := INT#1;
       GOTO Operator;
   END_IF;
END_REGION

REGION Network 32: Operating note 02: Service active / Bedienhinweis 02: Service aktiv
   // ATTRIBUT: 01 = BLUE / GREY (flashing Off) 02 = BLUE / GREY (flashing On) 03 = GREEN / GREY (flashing Off) 04 = GREEN / GREY (flashing On) 05 = RED / GREY (flashing off)06 = RED GREY (flashing On)07 = SW YELLOW (flashing Off) 08 = SW / YELLOW (flashing On) 09 = SW / ROT (flashing off) 10 = SW / RED (flashing On) 11 = SW / GREEN (flashing Off) 10 = SW / GREEN (flashing On)
   // ATTRIBUT: 01 = BLAU / GRAU (Blinken Aus)
   //           02 = BLAU / GRAU (Blinken Ein)
   //           03 = GRÜN / GRAU (Blinken Aus)
   //           04 = GRÜN / GRAU (Blinken Ein)
   //           05 = ROT  / GRAU (Blinken Aus)
   //           06 = ROT  / GRAU (Blinken Ein)
   //           07 = SW   / GELB (Blinken Aus)
   //           08 = SW   / GELB (Blinken Ein)
   //           09 = SW   / ROT  (Blinken Aus)
   //           10 = SW   / ROT  (Blinken Ein)
   //           11 = SW   / GRÜN (Blinken Aus)
   //           10 = SW   / GRÜN (Blinken Ein)
   RUNG wire#powerrail
      Contact( "AnwDB_OperatingModes_OP70".BA[0].mode_service )
      { S7_GenerateENO := "TRUE" } Move(in := INT#2, out1 => "LTLL_Data".HMI[0].global.prompt.index)
      { S7_GenerateENO := "TRUE" } Move(in := INT#8, out1 => "LTLL_Data".HMI[0].global.prompt.attribut)
      JumpCoil( Operator )
   END_RUNG
   // the same network as SCL:
   // ENO of a box is taken as its EN; it also drops when the box reports an error
   IF "AnwDB_OperatingModes_OP70".BA[0].mode_service THEN
       "LTLL_Data".HMI[0].global.prompt.index := INT#2;
       "LTLL_Data".HMI[0].global.prompt.attribut := INT#8;
       GOTO Operator;
   END_IF;
END_REGION

REGION Network 33: Operating note 03: Step mode active / Bedienhinweis 03: Schrittbetrieb aktiv
   // ATTRIBUT: 01 = BLUE / GREY (flashing Off) 02 = BLUE / GREY (flashing On) 03 = GREEN / GREY (flashing Off) 04 = GREEN / GREY (flashing On) 05 = RED / GREY (flashing off)06 = RED GREY (flashing On)07 = SW YELLOW (flashing Off) 08 = SW / YELLOW (flashing On) 09 = SW / ROT (flashing off) 10 = SW / RED (flashing On) 11 = SW / GREEN (flashing Off) 10 = SW / GREEN (flashing On)
   // ATTRIBUT: 01 = BLAU / GRAU (Blinken Aus)
   //           02 = BLAU / GRAU (Blinken Ein)
   //           03 = GRÜN / GRAU (Blinken Aus)
   //           04 = GRÜN / GRAU (Blinken Ein)
   //           05 = ROT  / GRAU (Blinken Aus)
   //           06 = ROT  / GRAU (Blinken Ein)
   //           07 = SW   / GELB (Blinken Aus)
   //           08 = SW   / GELB (Blinken Ein)
   //           09 = SW   / ROT  (Blinken Aus)
   //           10 = SW   / ROT  (Blinken Ein)
   //           11 = SW   / GRÜN (Blinken Aus)
   //           10 = SW   / GRÜN (Blinken Ein)
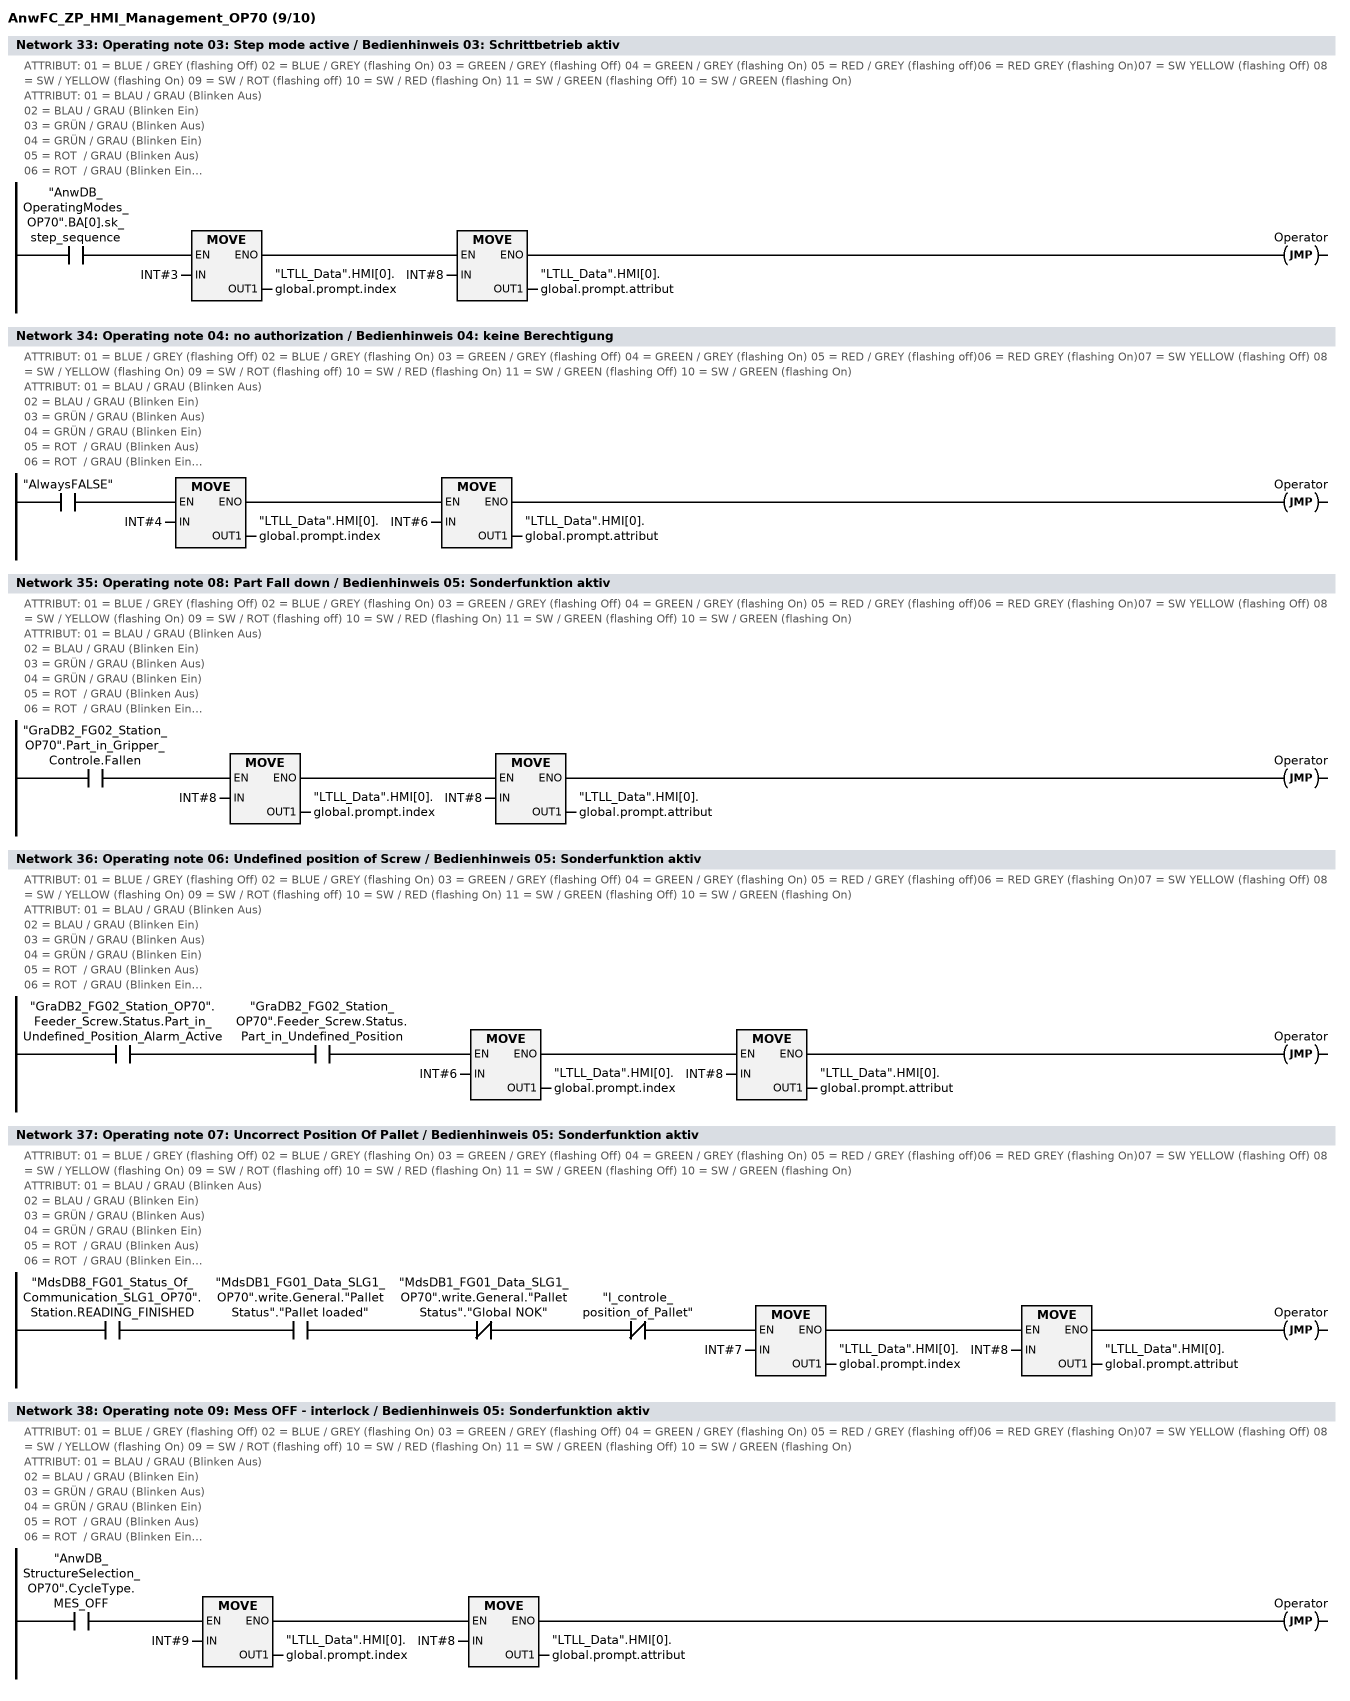
   RUNG wire#powerrail
      Contact( "AnwDB_OperatingModes_OP70".BA[0].sk_step_sequence )
      { S7_GenerateENO := "TRUE" } Move(in := INT#3, out1 => "LTLL_Data".HMI[0].global.prompt.index)
      { S7_GenerateENO := "TRUE" } Move(in := INT#8, out1 => "LTLL_Data".HMI[0].global.prompt.attribut)
      JumpCoil( Operator )
   END_RUNG
   // the same network as SCL:
   // ENO of a box is taken as its EN; it also drops when the box reports an error
   IF "AnwDB_OperatingModes_OP70".BA[0].sk_step_sequence THEN
       "LTLL_Data".HMI[0].global.prompt.index := INT#3;
       "LTLL_Data".HMI[0].global.prompt.attribut := INT#8;
       GOTO Operator;
   END_IF;
END_REGION

REGION Network 34: Operating note 04: no authorization / Bedienhinweis 04: keine Berechtigung
   // ATTRIBUT: 01 = BLUE / GREY (flashing Off) 02 = BLUE / GREY (flashing On) 03 = GREEN / GREY (flashing Off) 04 = GREEN / GREY (flashing On) 05 = RED / GREY (flashing off)06 = RED GREY (flashing On)07 = SW YELLOW (flashing Off) 08 = SW / YELLOW (flashing On) 09 = SW / ROT (flashing off) 10 = SW / RED (flashing On) 11 = SW / GREEN (flashing Off) 10 = SW / GREEN (flashing On)
   // ATTRIBUT: 01 = BLAU / GRAU (Blinken Aus)
   //           02 = BLAU / GRAU (Blinken Ein)
   //           03 = GRÜN / GRAU (Blinken Aus)
   //           04 = GRÜN / GRAU (Blinken Ein)
   //           05 = ROT  / GRAU (Blinken Aus)
   //           06 = ROT  / GRAU (Blinken Ein)
   //           07 = SW   / GELB (Blinken Aus)
   //           08 = SW   / GELB (Blinken Ein)
   //           09 = SW   / ROT  (Blinken Aus)
   //           10 = SW   / ROT  (Blinken Ein)
   //           11 = SW   / GRÜN (Blinken Aus)
   //           10 = SW   / GRÜN (Blinken Ein)
   RUNG wire#powerrail
      Contact( "AlwaysFALSE" )
      { S7_GenerateENO := "TRUE" } Move(in := INT#4, out1 => "LTLL_Data".HMI[0].global.prompt.index)
      { S7_GenerateENO := "TRUE" } Move(in := INT#6, out1 => "LTLL_Data".HMI[0].global.prompt.attribut)
      JumpCoil( Operator )
   END_RUNG
   // the same network as SCL:
   // ENO of a box is taken as its EN; it also drops when the box reports an error
   IF "AlwaysFALSE" THEN
       "LTLL_Data".HMI[0].global.prompt.index := INT#4;
       "LTLL_Data".HMI[0].global.prompt.attribut := INT#6;
       GOTO Operator;
   END_IF;
END_REGION

REGION Network 35: Operating note 08: Part Fall down / Bedienhinweis 05: Sonderfunktion aktiv
   // ATTRIBUT: 01 = BLUE / GREY (flashing Off) 02 = BLUE / GREY (flashing On) 03 = GREEN / GREY (flashing Off) 04 = GREEN / GREY (flashing On) 05 = RED / GREY (flashing off)06 = RED GREY (flashing On)07 = SW YELLOW (flashing Off) 08 = SW / YELLOW (flashing On) 09 = SW / ROT (flashing off) 10 = SW / RED (flashing On) 11 = SW / GREEN (flashing Off) 10 = SW / GREEN (flashing On)
   // ATTRIBUT: 01 = BLAU / GRAU (Blinken Aus)
   //           02 = BLAU / GRAU (Blinken Ein)
   //           03 = GRÜN / GRAU (Blinken Aus)
   //           04 = GRÜN / GRAU (Blinken Ein)
   //           05 = ROT  / GRAU (Blinken Aus)
   //           06 = ROT  / GRAU (Blinken Ein)
   //           07 = SW   / GELB (Blinken Aus)
   //           08 = SW   / GELB (Blinken Ein)
   //           09 = SW   / ROT  (Blinken Aus)
   //           10 = SW   / ROT  (Blinken Ein)
   //           11 = SW   / GRÜN (Blinken Aus)
   //           10 = SW   / GRÜN (Blinken Ein)
   RUNG wire#powerrail
      Contact( "GraDB2_FG02_Station_OP70".Part_in_Gripper_Controle.Fallen )
      { S7_GenerateENO := "TRUE" } Move(in := INT#8, out1 => "LTLL_Data".HMI[0].global.prompt.index)
      { S7_GenerateENO := "TRUE" } Move(in := INT#8, out1 => "LTLL_Data".HMI[0].global.prompt.attribut)
      JumpCoil( Operator )
   END_RUNG
   // the same network as SCL:
   // ENO of a box is taken as its EN; it also drops when the box reports an error
   IF "GraDB2_FG02_Station_OP70".Part_in_Gripper_Controle.Fallen THEN
       "LTLL_Data".HMI[0].global.prompt.index := INT#8;
       "LTLL_Data".HMI[0].global.prompt.attribut := INT#8;
       GOTO Operator;
   END_IF;
END_REGION

REGION Network 36: Operating note 06: Undefined position of Screw / Bedienhinweis 05: Sonderfunktion aktiv
   // ATTRIBUT: 01 = BLUE / GREY (flashing Off) 02 = BLUE / GREY (flashing On) 03 = GREEN / GREY (flashing Off) 04 = GREEN / GREY (flashing On) 05 = RED / GREY (flashing off)06 = RED GREY (flashing On)07 = SW YELLOW (flashing Off) 08 = SW / YELLOW (flashing On) 09 = SW / ROT (flashing off) 10 = SW / RED (flashing On) 11 = SW / GREEN (flashing Off) 10 = SW / GREEN (flashing On)
   // ATTRIBUT: 01 = BLAU / GRAU (Blinken Aus)
   //           02 = BLAU / GRAU (Blinken Ein)
   //           03 = GRÜN / GRAU (Blinken Aus)
   //           04 = GRÜN / GRAU (Blinken Ein)
   //           05 = ROT  / GRAU (Blinken Aus)
   //           06 = ROT  / GRAU (Blinken Ein)
   //           07 = SW   / GELB (Blinken Aus)
   //           08 = SW   / GELB (Blinken Ein)
   //           09 = SW   / ROT  (Blinken Aus)
   //           10 = SW   / ROT  (Blinken Ein)
   //           11 = SW   / GRÜN (Blinken Aus)
   //           10 = SW   / GRÜN (Blinken Ein)
   RUNG wire#powerrail
      Contact( "GraDB2_FG02_Station_OP70".Feeder_Screw.Status.Part_in_Undefined_Position_Alarm_Active )
      Contact( "GraDB2_FG02_Station_OP70".Feeder_Screw.Status.Part_in_Undefined_Position )
      { S7_GenerateENO := "TRUE" } Move(in := INT#6, out1 => "LTLL_Data".HMI[0].global.prompt.index)
      { S7_GenerateENO := "TRUE" } Move(in := INT#8, out1 => "LTLL_Data".HMI[0].global.prompt.attribut)
      JumpCoil( Operator )
   END_RUNG
   // the same network as SCL:
   // ENO of a box is taken as its EN; it also drops when the box reports an error
   #_w1 := "GraDB2_FG02_Station_OP70".Feeder_Screw.Status.Part_in_Undefined_Position_Alarm_Active AND "GraDB2_FG02_Station_OP70".Feeder_Screw.Status.Part_in_Undefined_Position;
   IF #_w1 THEN
       "LTLL_Data".HMI[0].global.prompt.index := INT#6;
       "LTLL_Data".HMI[0].global.prompt.attribut := INT#8;
       GOTO Operator;
   END_IF;
END_REGION

REGION Network 37: Operating note 07: Uncorrect Position Of Pallet / Bedienhinweis 05: Sonderfunktion aktiv
   // ATTRIBUT: 01 = BLUE / GREY (flashing Off) 02 = BLUE / GREY (flashing On) 03 = GREEN / GREY (flashing Off) 04 = GREEN / GREY (flashing On) 05 = RED / GREY (flashing off)06 = RED GREY (flashing On)07 = SW YELLOW (flashing Off) 08 = SW / YELLOW (flashing On) 09 = SW / ROT (flashing off) 10 = SW / RED (flashing On) 11 = SW / GREEN (flashing Off) 10 = SW / GREEN (flashing On)
   // ATTRIBUT: 01 = BLAU / GRAU (Blinken Aus)
   //           02 = BLAU / GRAU (Blinken Ein)
   //           03 = GRÜN / GRAU (Blinken Aus)
   //           04 = GRÜN / GRAU (Blinken Ein)
   //           05 = ROT  / GRAU (Blinken Aus)
   //           06 = ROT  / GRAU (Blinken Ein)
   //           07 = SW   / GELB (Blinken Aus)
   //           08 = SW   / GELB (Blinken Ein)
   //           09 = SW   / ROT  (Blinken Aus)
   //           10 = SW   / ROT  (Blinken Ein)
   //           11 = SW   / GRÜN (Blinken Aus)
   //           10 = SW   / GRÜN (Blinken Ein)
   RUNG wire#powerrail
      Contact( "MdsDB8_FG01_Status_Of_Communication_SLG1_OP70".Station.READING_FINISHED )
      Contact( "MdsDB1_FG01_Data_SLG1_OP70".write.General."Pallet Status"."Pallet loaded" )
      I_Contact( "MdsDB1_FG01_Data_SLG1_OP70".write.General."Pallet Status"."Global NOK" )
      I_Contact( "I_controle_position_of_Pallet" )
      { S7_GenerateENO := "TRUE" } Move(in := INT#7, out1 => "LTLL_Data".HMI[0].global.prompt.index)
      { S7_GenerateENO := "TRUE" } Move(in := INT#8, out1 => "LTLL_Data".HMI[0].global.prompt.attribut)
      JumpCoil( Operator )
   END_RUNG
   // the same network as SCL:
   // ENO of a box is taken as its EN; it also drops when the box reports an error
   #_w1 := "MdsDB8_FG01_Status_Of_Communication_SLG1_OP70".Station.READING_FINISHED AND "MdsDB1_FG01_Data_SLG1_OP70".write.General."Pallet Status"."Pallet loaded" AND NOT "MdsDB1_FG01_Data_SLG1_OP70".write.General."Pallet Status"."Global NOK" AND NOT "I_controle_position_of_Pallet";
   IF #_w1 THEN
       "LTLL_Data".HMI[0].global.prompt.index := INT#7;
       "LTLL_Data".HMI[0].global.prompt.attribut := INT#8;
       GOTO Operator;
   END_IF;
END_REGION

REGION Network 38: Operating note 09: Mess OFF - interlock / Bedienhinweis 05: Sonderfunktion aktiv
   // ATTRIBUT: 01 = BLUE / GREY (flashing Off) 02 = BLUE / GREY (flashing On) 03 = GREEN / GREY (flashing Off) 04 = GREEN / GREY (flashing On) 05 = RED / GREY (flashing off)06 = RED GREY (flashing On)07 = SW YELLOW (flashing Off) 08 = SW / YELLOW (flashing On) 09 = SW / ROT (flashing off) 10 = SW / RED (flashing On) 11 = SW / GREEN (flashing Off) 10 = SW / GREEN (flashing On)
   // ATTRIBUT: 01 = BLAU / GRAU (Blinken Aus)
   //           02 = BLAU / GRAU (Blinken Ein)
   //           03 = GRÜN / GRAU (Blinken Aus)
   //           04 = GRÜN / GRAU (Blinken Ein)
   //           05 = ROT  / GRAU (Blinken Aus)
   //           06 = ROT  / GRAU (Blinken Ein)
   //           07 = SW   / GELB (Blinken Aus)
   //           08 = SW   / GELB (Blinken Ein)
   //           09 = SW   / ROT  (Blinken Aus)
   //           10 = SW   / ROT  (Blinken Ein)
   //           11 = SW   / GRÜN (Blinken Aus)
   //           10 = SW   / GRÜN (Blinken Ein)
   RUNG wire#powerrail
      Contact( "AnwDB_StructureSelection_OP70".CycleType.MES_OFF )
      { S7_GenerateENO := "TRUE" } Move(in := INT#9, out1 => "LTLL_Data".HMI[0].global.prompt.index)
      { S7_GenerateENO := "TRUE" } Move(in := INT#8, out1 => "LTLL_Data".HMI[0].global.prompt.attribut)
      JumpCoil( Operator )
   END_RUNG
   // the same network as SCL:
   // ENO of a box is taken as its EN; it also drops when the box reports an error
   IF "AnwDB_StructureSelection_OP70".CycleType.MES_OFF THEN
       "LTLL_Data".HMI[0].global.prompt.index := INT#9;
       "LTLL_Data".HMI[0].global.prompt.attribut := INT#8;
       GOTO Operator;
   END_IF;
END_REGION

REGION Network 39: Operating note 10: Mess OFF - Tracibility
   // ATTRIBUT: 01 = BLUE / GREY (flashing Off) 02 = BLUE / GREY (flashing On) 03 = GREEN / GREY (flashing Off) 04 = GREEN / GREY (flashing On) 05 = RED / GREY (flashing off)06 = RED GREY (flashing On)07 = SW YELLOW (flashing Off) 08 = SW / YELLOW (flashing On) 09 = SW / ROT (flashing off) 10 = SW / RED (flashing On) 11 = SW / GREEN (flashing Off) 10 = SW / GREEN (flashing On)
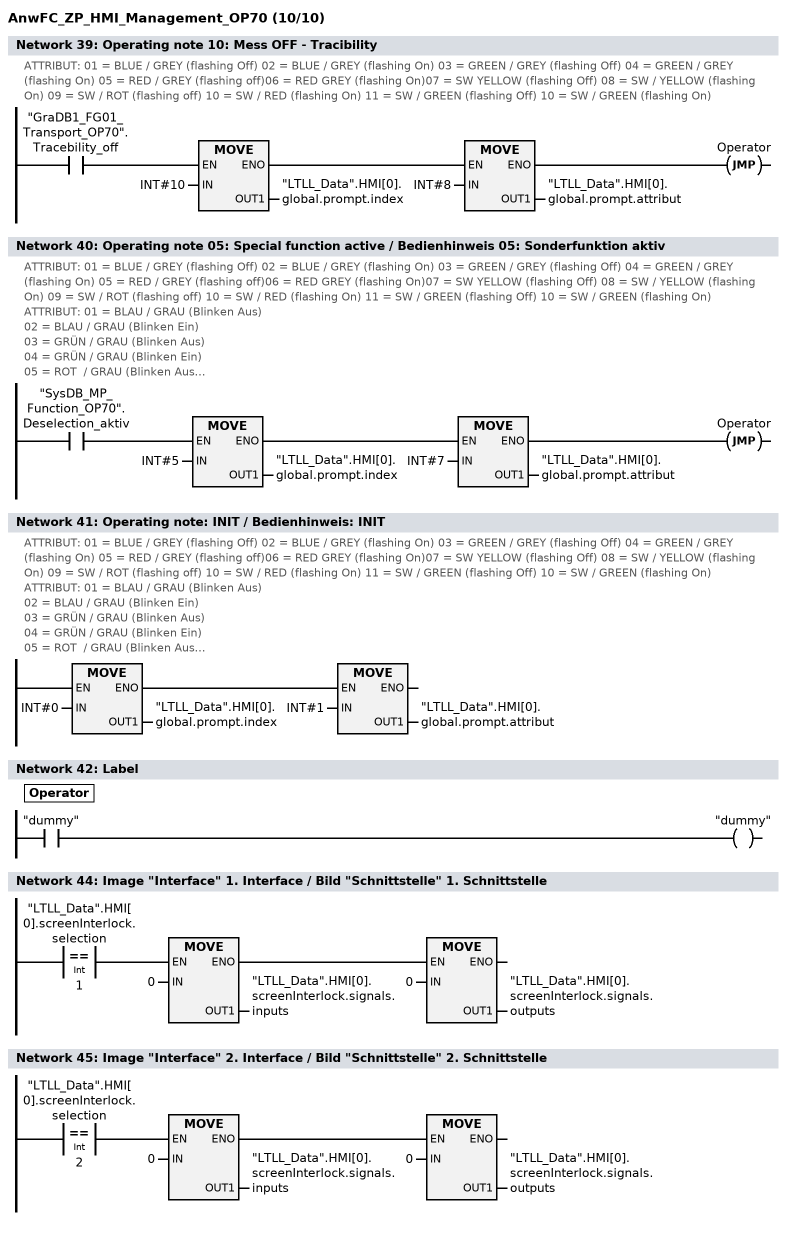
   RUNG wire#powerrail
      Contact( "GraDB1_FG01_Transport_OP70".Tracebility_off )
      { S7_GenerateENO := "TRUE" } Move(in := INT#10, out1 => "LTLL_Data".HMI[0].global.prompt.index)
      { S7_GenerateENO := "TRUE" } Move(in := INT#8, out1 => "LTLL_Data".HMI[0].global.prompt.attribut)
      JumpCoil( Operator )
   END_RUNG
   // the same network as SCL:
   // ENO of a box is taken as its EN; it also drops when the box reports an error
   IF "GraDB1_FG01_Transport_OP70".Tracebility_off THEN
       "LTLL_Data".HMI[0].global.prompt.index := INT#10;
       "LTLL_Data".HMI[0].global.prompt.attribut := INT#8;
       GOTO Operator;
   END_IF;
END_REGION

REGION Network 40: Operating note 05: Special function active / Bedienhinweis 05: Sonderfunktion aktiv
   // ATTRIBUT: 01 = BLUE / GREY (flashing Off) 02 = BLUE / GREY (flashing On) 03 = GREEN / GREY (flashing Off) 04 = GREEN / GREY (flashing On) 05 = RED / GREY (flashing off)06 = RED GREY (flashing On)07 = SW YELLOW (flashing Off) 08 = SW / YELLOW (flashing On) 09 = SW / ROT (flashing off) 10 = SW / RED (flashing On) 11 = SW / GREEN (flashing Off) 10 = SW / GREEN (flashing On)
   // ATTRIBUT: 01 = BLAU / GRAU (Blinken Aus)
   //           02 = BLAU / GRAU (Blinken Ein)
   //           03 = GRÜN / GRAU (Blinken Aus)
   //           04 = GRÜN / GRAU (Blinken Ein)
   //           05 = ROT  / GRAU (Blinken Aus)
   //           06 = ROT  / GRAU (Blinken Ein)
   //           07 = SW   / GELB (Blinken Aus)
   //           08 = SW   / GELB (Blinken Ein)
   //           09 = SW   / ROT  (Blinken Aus)
   //           10 = SW   / ROT  (Blinken Ein)
   //           11 = SW   / GRÜN (Blinken Aus)
   //           10 = SW   / GRÜN (Blinken Ein)
   RUNG wire#powerrail
      Contact( "SysDB_MP_Function_OP70".Deselection_aktiv )
      { S7_GenerateENO := "TRUE" } Move(in := INT#5, out1 => "LTLL_Data".HMI[0].global.prompt.index)
      { S7_GenerateENO := "TRUE" } Move(in := INT#7, out1 => "LTLL_Data".HMI[0].global.prompt.attribut)
      JumpCoil( Operator )
   END_RUNG
   // the same network as SCL:
   // ENO of a box is taken as its EN; it also drops when the box reports an error
   IF "SysDB_MP_Function_OP70".Deselection_aktiv THEN
       "LTLL_Data".HMI[0].global.prompt.index := INT#5;
       "LTLL_Data".HMI[0].global.prompt.attribut := INT#7;
       GOTO Operator;
   END_IF;
END_REGION

REGION Network 41: Operating note: INIT / Bedienhinweis: INIT
   // ATTRIBUT: 01 = BLUE / GREY (flashing Off) 02 = BLUE / GREY (flashing On) 03 = GREEN / GREY (flashing Off) 04 = GREEN / GREY (flashing On) 05 = RED / GREY (flashing off)06 = RED GREY (flashing On)07 = SW YELLOW (flashing Off) 08 = SW / YELLOW (flashing On) 09 = SW / ROT (flashing off) 10 = SW / RED (flashing On) 11 = SW / GREEN (flashing Off) 10 = SW / GREEN (flashing On)
   // ATTRIBUT: 01 = BLAU / GRAU (Blinken Aus)
   //           02 = BLAU / GRAU (Blinken Ein)
   //           03 = GRÜN / GRAU (Blinken Aus)
   //           04 = GRÜN / GRAU (Blinken Ein)
   //           05 = ROT  / GRAU (Blinken Aus)
   //           06 = ROT  / GRAU (Blinken Ein)
   //           07 = SW   / GELB (Blinken Aus)
   //           08 = SW   / GELB (Blinken Ein)
   //           09 = SW   / ROT  (Blinken Aus)
   //           10 = SW   / ROT  (Blinken Ein)
   //           11 = SW   / GRÜN (Blinken Aus)
   //           10 = SW   / GRÜN (Blinken Ein)
   RUNG wire#powerrail
      { S7_GenerateENO := "TRUE" } Move(in := INT#0, out1 => "LTLL_Data".HMI[0].global.prompt.index)
      { S7_GenerateENO := "TRUE" } Move(in := INT#1, out1 => "LTLL_Data".HMI[0].global.prompt.attribut)
   END_RUNG
   // the same network as SCL:
   // ENO of a box is taken as its EN; it also drops when the box reports an error
   "LTLL_Data".HMI[0].global.prompt.index := INT#0;
   "LTLL_Data".HMI[0].global.prompt.attribut := INT#1;
END_REGION

REGION Network 42: Label
   Label( Operator )
   RUNG wire#powerrail
      Contact( "dummy" )
      Coil( "dummy" )
   END_RUNG
   // the same network as SCL:
   Operator:
   "dummy" := "dummy";
END_REGION

REGION Network 43: ############# SS_04_031_Interlocks ############## / ########################### SS_04_031_Interlocks #############################
END_REGION

REGION Network 44: Image "Interface" 1. Interface / Bild "Schnittstelle" 1. Schnittstelle
   RUNG wire#powerrail
      { S7_Templates := "SrcType := Int" } EQ_Contact(in1 := "LTLL_Data".HMI[0].screenInterlock.selection, in2 := 1)
      { S7_GenerateENO := "TRUE" } Move(in := 0, out1 => "LTLL_Data".HMI[0].screenInterlock.signals.inputs)
      { S7_GenerateENO := "TRUE" } Move(in := 0, out1 => "LTLL_Data".HMI[0].screenInterlock.signals.outputs)
   END_RUNG
   // the same network as SCL:
   // ENO of a box is taken as its EN; it also drops when the box reports an error
   #_w1 := "LTLL_Data".HMI[0].screenInterlock.selection = 1;
   IF #_w1 THEN
       "LTLL_Data".HMI[0].screenInterlock.signals.inputs := 0;
       "LTLL_Data".HMI[0].screenInterlock.signals.outputs := 0;
   END_IF;
END_REGION

REGION Network 45: Image "Interface" 2. Interface / Bild "Schnittstelle" 2. Schnittstelle
   RUNG wire#powerrail
      { S7_Templates := "SrcType := Int" } EQ_Contact(in1 := "LTLL_Data".HMI[0].screenInterlock.selection, in2 := 2)
      { S7_GenerateENO := "TRUE" } Move(in := 0, out1 => "LTLL_Data".HMI[0].screenInterlock.signals.inputs)
      { S7_GenerateENO := "TRUE" } Move(in := 0, out1 => "LTLL_Data".HMI[0].screenInterlock.signals.outputs)
   END_RUNG
   // the same network as SCL:
   // ENO of a box is taken as its EN; it also drops when the box reports an error
   #_w1 := "LTLL_Data".HMI[0].screenInterlock.selection = 2;
   IF #_w1 THEN
       "LTLL_Data".HMI[0].screenInterlock.signals.inputs := 0;
       "LTLL_Data".HMI[0].screenInterlock.signals.outputs := 0;
   END_IF;
END_REGION

REGION Network 46: END / ENDE
END_REGION
END_FUNCTION
